LIN {X 0,Y 474.618,Z 150.861,A -85,B 0,C 180,E1 -7365.42,E2 -7365.42} C_VEL
LIN {X 0,Y 474.69,Z 150.851,A -85,B 0,C 180,E1 -7368.037,E2 -7368.037} C_VEL
LIN {X 0,Y 474.695,Z 150.851,A -85,B 0,C 180,E1 -7371.486,E2 -7371.486} C_VEL
LIN {X 0,Y 474.744,Z 150.845,A -85,B 0,C 180,E1 -7374.052,E2 -7374.052} C_VEL
LIN {X 0,Y 474.866,Z 150.829,A -85,B 0,C 180,E1 -7377.455,E2 -7377.455} C_VEL
LIN {X 0,Y 474.862,Z 150.83,A -85,B 0,C 180,E1 -7380,E2 -7380} C_VEL
LIN {X 0,Y 474.862,Z 150.835,A -85,B 0,C 180,E1 -7382.544,E2 -7382.544} C_VEL
LIN {X 0,Y 474.742,Z 150.847,A -85,B 0,C 180,E1 -7385.948,E2 -7385.948} C_VEL
LIN {X 0,Y 474.685,Z 150.857,A -85,B 0,C 180,E1 -7388.514,E2 -7388.514} C_VEL
LIN {X 0,Y 474.677,Z 150.856,A -85,B 0,C 180,E1 -7391.963,E2 -7391.963} C_VEL
LIN {X 0,Y 474.683,Z 150.854,A -85,B 0,C 180,E1 -7395.456,E2 -7395.456} C_VEL
LIN {X 0,Y 474.646,Z 150.859,A -85,B 0,C 180,E1 -7399.011,E2 -7399.011} C_VEL
LIN {X 0,Y 474.574,Z 150.87,A -85,B 0,C 180,E1 -7401.729,E2 -7401.729} C_VEL
LIN {X 0,Y 474.611,Z 150.865,A -85,B 0,C 180,E1 -7404.495,E2 -7404.495} C_VEL
LIN {X 0,Y 474.583,Z 150.867,A -85,B 0,C 180,E1 -7407.327,E2 -7407.327} C_VEL
LIN {X 0,Y 474.596,Z 150.87,A -85,B 0,C 180,E1 -7410.23,E2 -7410.23} C_VEL
LIN {X 0,Y 474.648,Z 151.03,A -85,B 0,C 180,E1 -7411.586,E2 -7411.586} C_VEL
LIN {X 0,Y 475.967,Z 158.401,A -85,B 0,C 180,E1 -7413.115,E2 -7413.115} C_VEL
LIN {X 0,Y 475.697,Z 171.558,A -85,B 0,C 180,E1 -7415.654,E2 -7415.654} C_VEL
LIN {X 0,Y 475.449,Z 180.026,A -85,B 0,C 180,E1 -7417.232,E2 -7417.232} C_VEL
LIN {X 0,Y 476.208,Z 184.236,A -85,B 0,C 180,E1 -7417.368,E2 -7417.368} C_VEL
LIN {X 0,Y 478.194,Z 196.098,A -85,B 0,C 180,E1 -7417.633,E2 -7417.633} C_VEL
LIN {X 0,Y 477.381,Z 287.664,A -85,B 0,C 180,E1 -7419.069,E2 -7419.069} C_VEL
LIN {X 0,Y 477.141,Z 300.656,A -85,B 0,C 180,E1 -7419.44,E2 -7419.44} C_VEL
LIN {X 0,Y 476.759,Z 313.013,A -85,B 0,C 180,E1 -7419.958,E2 -7419.958} C_VEL
LIN {X 0,Y 476.372,Z 324.473,A -85,B 0,C 180,E1 -7420.606,E2 -7420.606} C_VEL
LIN {X 0,Y 475.88,Z 335.964,A -85,B 0,C 180,E1 -7421.447,E2 -7421.447} C_VEL
LIN {X 0,Y 475.436,Z 345.842,A -85,B 0,C 180,E1 -7422.347,E2 -7422.347} C_VEL
LIN {X 0,Y 475.017,Z 354.974,A -85,B 0,C 180,E1 -7423.363,E2 -7423.363} C_VEL
LIN {X 0,Y 474.602,Z 363.651,A -85,B 0,C 180,E1 -7424.545,E2 -7424.545} C_VEL
LIN {X 0,Y 474.265,Z 371.371,A -85,B 0,C 180,E1 -7425.857,E2 -7425.857} C_VEL
LIN {X 0,Y 474.065,Z 376.86,A -85,B 0,C 180,E1 -7427.006,E2 -7427.006} C_VEL
LIN {X 0,Y 473.921,Z 381.283,A -85,B 0,C 180,E1 -7428.141,E2 -7428.141} C_VEL
LIN {X 0,Y 473.859,Z 384.78,A -85,B 0,C 180,E1 -7429.265,E2 -7429.265} C_VEL
LIN {X 0,Y 473.679,Z 387.66,A -85,B 0,C 180,E1 -7430.49,E2 -7430.49} C_VEL
LIN {X 0,Y 473.595,Z 389.84,A -85,B 0,C 180,E1 -7431.859,E2 -7431.859} C_VEL
LIN {X 0,Y 473.572,Z 390.497,A -85,B 0,C 180,E1 -7432.508,E2 -7432.508} C_VEL
LIN {X 0,Y 472.915,Z 391.073,A -85,B 0,C 180,E1 -7433.216,E2 -7433.216} C_VEL
LIN {X 0,Y 470.061,Z 391.361,A -85,B 0,C 180,E1 -7434.371,E2 -7434.371} C_VEL
LIN {X 0,Y 467.642,Z 390.943,A -85,B 0,C 180,E1 -7435.301,E2 -7435.301} C_VEL
LIN {X 0,Y 466.601,Z 390.22,A -85,B 0,C 180,E1 -7436.015,E2 -7436.015} C_VEL
LIN {X 0,Y 466.515,Z 389.897,A -85,B 0,C 180,E1 -7436.255,E2 -7436.255} C_VEL
LIN {X 0,Y 466.607,Z 387.998,A -85,B 0,C 180,E1 -7437.507,E2 -7437.507} C_VEL
LIN {X 0,Y 466.734,Z 384.141,A -85,B 0,C 180,E1 -7439.125,E2 -7439.125} C_VEL
LIN {X 0,Y 466.909,Z 379.431,A -85,B 0,C 180,E1 -7440.543,E2 -7440.543} C_VEL
LIN {X 0,Y 467.152,Z 373.328,A -85,B 0,C 180,E1 -7441.958,E2 -7441.958} C_VEL
LIN {X 0,Y 467.413,Z 366.653,A -85,B 0,C 180,E1 -7443.189,E2 -7443.189} C_VEL
LIN {X 0,Y 467.847,Z 357.754,A -85,B 0,C 180,E1 -7444.505,E2 -7444.505} C_VEL
LIN {X 0,Y 468.279,Z 348.414,A -85,B 0,C 180,E1 -7445.625,E2 -7445.625} C_VEL
LIN {X 0,Y 468.758,Z 338.491,A -85,B 0,C 180,E1 -7446.591,E2 -7446.591} C_VEL
LIN {X 0,Y 469.247,Z 327.717,A -85,B 0,C 180,E1 -7447.433,E2 -7447.433} C_VEL
LIN {X 0,Y 469.72,Z 315.436,A -85,B 0,C 180,E1 -7448.185,E2 -7448.185} C_VEL
LIN {X 0,Y 470.111,Z 303.17,A -85,B 0,C 180,E1 -7448.746,E2 -7448.746} C_VEL
LIN {X 0,Y 470.403,Z 289.73,A -85,B 0,C 180,E1 -7449.161,E2 -7449.161} C_VEL
LIN {X 0,Y 470.644,Z 267.567,A -85,B 0,C 180,E1 -7449.543,E2 -7449.543} C_VEL
LIN {X 0,Y 471.141,Z 195.55,A -85,B 0,C 180,E1 -7450.672,E2 -7450.672} C_VEL
LIN {X 0,Y 468.481,Z 180.547,A -85,B 0,C 180,E1 -7451.028,E2 -7451.028} C_VEL
LIN {X 0,Y 468.525,Z 177.121,A -85,B 0,C 180,E1 -7451.64,E2 -7451.64} C_VEL
LIN {X 0,Y 469.221,Z 161.481,A -85,B 0,C 180,E1 -7454.806,E2 -7454.806} C_VEL
LIN {X 0,Y 468.327,Z 155.391,A -85,B 0,C 180,E1 -7456.108,E2 -7456.108} C_VEL
LIN {X 0,Y 467.639,Z 151.805,A -85,B 0,C 180,E1 -7456.945,E2 -7456.945} C_VEL
LIN {X 0,Y 467.624,Z 151.736,A -85,B 0,C 180,E1 -7459.611,E2 -7459.611} C_VEL
LIN {X 0,Y 467.749,Z 151.716,A -85,B 0,C 180,E1 -7462.591,E2 -7462.591} C_VEL
LIN {X 0,Y 467.721,Z 151.719,A -85,B 0,C 180,E1 -7464.828,E2 -7464.828} C_VEL
LIN {X 0,Y 467.856,Z 151.705,A -85,B 0,C 180,E1 -7467.418,E2 -7467.418} C_VEL
LIN {X 0,Y 467.879,Z 151.704,A -85,B 0,C 180,E1 -7470.001,E2 -7470.001} C_VEL
LIN {X 0,Y 467.856,Z 151.702,A -85,B 0,C 180,E1 -7472.584,E2 -7472.584} C_VEL
LIN {X 0,Y 467.732,Z 151.721,A -85,B 0,C 180,E1 -7476.038,E2 -7476.038} C_VEL
LIN {X 0,Y 467.669,Z 151.726,A -85,B 0,C 180,E1 -7478.644,E2 -7478.644} C_VEL
LIN {X 0,Y 467.655,Z 151.728,A -85,B 0,C 180,E1 -7482.146,E2 -7482.146} C_VEL
LIN {X 0,Y 467.638,Z 151.734,A -85,B 0,C 180,E1 -7485.696,E2 -7485.696} C_VEL
LIN {X 0,Y 467.621,Z 151.74,A -85,B 0,C 180,E1 -7489.308,E2 -7489.308} C_VEL
LIN {X 0,Y 467.533,Z 151.743,A -85,B 0,C 180,E1 -7492.075,E2 -7492.075} C_VEL
LIN {X 0,Y 467.584,Z 151.74,A -85,B 0,C 180,E1 -7494.889,E2 -7494.889} C_VEL
LIN {X 0,Y 467.618,Z 151.733,A -85,B 0,C 180,E1 -7497.77,E2 -7497.77} C_VEL
LIN {X 0,Y 467.566,Z 151.746,A -85,B 0,C 180,E1 -7501.045,E2 -7501.045} C_VEL
LIN {X 0,Y 467.576,Z 151.738,A -85,B 0,C 180,E1 -7504.241,E2 -7504.241} C_VEL
LIN {X 0,Y 467.547,Z 151.746,A -85,B 0,C 180,E1 -7507.187,E2 -7507.187} C_VEL
LIN {X 0,Y 467.573,Z 151.739,A -85,B 0,C 180,E1 -7510.265,E2 -7510.265} C_VEL
LIN {X 0,Y 467.586,Z 151.741,A -85,B 0,C 180,E1 -7512.567,E2 -7512.567} C_VEL
LIN {X 0,Y 467.565,Z 151.743,A -85,B 0,C 180,E1 -7515.053,E2 -7515.053} C_VEL
LIN {X 0,Y 467.572,Z 151.745,A -85,B 0,C 180,E1 -7518.597,E2 -7518.597} C_VEL
LIN {X 0,Y 467.561,Z 151.74,A -85,B 0,C 180,E1 -7521.956,E2 -7521.956} C_VEL
LIN {X 0,Y 467.561,Z 151.74,A -85,B 0,C 180,E1 -7525.168,E2 -7525.168} C_VEL
LIN {X 0,Y 467.582,Z 151.742,A -85,B 0,C 180,E1 -7528.26,E2 -7528.26} C_VEL
LIN {X 0,Y 467.554,Z 151.74,A -85,B 0,C 180,E1 -7531.249,E2 -7531.249} C_VEL
LIN {X 0,Y 467.582,Z 151.742,A -85,B 0,C 180,E1 -7534.159,E2 -7534.159} C_VEL
LIN {X 0,Y 467.575,Z 151.738,A -85,B 0,C 180,E1 -7536.996,E2 -7536.996} C_VEL
LIN {X 0,Y 467.621,Z 151.734,A -85,B 0,C 180,E1 -7539.778,E2 -7539.778} C_VEL
LIN {X 0,Y 467.593,Z 151.739,A -85,B 0,C 180,E1 -7542.507,E2 -7542.507} C_VEL
LIN {X 0,Y 467.599,Z 151.734,A -85,B 0,C 180,E1 -7545.197,E2 -7545.197} C_VEL
LIN {X 0,Y 467.656,Z 151.733,A -85,B 0,C 180,E1 -7547.855,E2 -7547.855} C_VEL
LIN {X 0,Y 467.657,Z 151.728,A -85,B 0,C 180,E1 -7551.357,E2 -7551.357} C_VEL
LIN {X 0,Y 467.702,Z 151.729,A -85,B 0,C 180,E1 -7553.962,E2 -7553.962} C_VEL
LIN {X 0,Y 467.813,Z 151.71,A -85,B 0,C 180,E1 -7557.417,E2 -7557.417} C_VEL
LIN {X 0,Y 467.848,Z 151.708,A -85,B 0,C 180,E1 -7560,E2 -7560} C_VEL
LIN {X 0,Y 467.822,Z 151.707,A -85,B 0,C 180,E1 -7562.583,E2 -7562.583} C_VEL
LIN {X 0,Y 467.694,Z 151.726,A -85,B 0,C 180,E1 -7566.038,E2 -7566.038} C_VEL
LIN {X 0,Y 467.636,Z 151.73,A -85,B 0,C 180,E1 -7568.644,E2 -7568.644} C_VEL
LIN {X 0,Y 467.656,Z 151.728,A -85,B 0,C 180,E1 -7572.146,E2 -7572.146} C_VEL
LIN {X 0,Y 467.638,Z 151.734,A -85,B 0,C 180,E1 -7575.695,E2 -7575.695} C_VEL
LIN {X 0,Y 467.617,Z 151.74,A -85,B 0,C 180,E1 -7579.308,E2 -7579.308} C_VEL
LIN {X 0,Y 467.53,Z 151.743,A -85,B 0,C 180,E1 -7582.074,E2 -7582.074} C_VEL
LIN {X 0,Y 467.551,Z 151.744,A -85,B 0,C 180,E1 -7584.891,E2 -7584.891} C_VEL
LIN {X 0,Y 467.538,Z 151.743,A -85,B 0,C 180,E1 -7587.775,E2 -7587.775} C_VEL
LIN {X 0,Y 467.528,Z 151.75,A -85,B 0,C 180,E1 -7591.036,E2 -7591.036} C_VEL
LIN {X 0,Y 467.566,Z 151.739,A -85,B 0,C 180,E1 -7594.238,E2 -7594.238} C_VEL
LIN {X 0,Y 467.517,Z 151.75,A -85,B 0,C 180,E1 -7597.181,E2 -7597.181} C_VEL
LIN {X 0,Y 467.519,Z 151.745,A -85,B 0,C 180,E1 -7600.271,E2 -7600.271} C_VEL
LIN {X 0,Y 467.518,Z 151.749,A -85,B 0,C 180,E1 -7602.569,E2 -7602.569} C_VEL
LIN {X 0,Y 467.564,Z 151.743,A -85,B 0,C 180,E1 -7605.052,E2 -7605.052} C_VEL
LIN {X 0,Y 467.552,Z 151.748,A -85,B 0,C 180,E1 -7608.727,E2 -7608.727} C_VEL
LIN {X 0,Y 467.533,Z 151.743,A -85,B 0,C 180,E1 -7611.952,E2 -7611.952} C_VEL
LIN {X 0,Y 467.511,Z 151.747,A -85,B 0,C 180,E1 -7615.162,E2 -7615.162} C_VEL
LIN {X 0,Y 467.544,Z 151.746,A -85,B 0,C 180,E1 -7618.256,E2 -7618.256} C_VEL
LIN {X 0,Y 467.527,Z 151.747,A -85,B 0,C 180,E1 -7621.247,E2 -7621.247} C_VEL
LIN {X 0,Y 467.571,Z 151.743,A -85,B 0,C 180,E1 -7624.693,E2 -7624.693} C_VEL
LIN {X 0,Y 467.652,Z 152.044,A -85,B 0,C 180,E1 -7625.063,E2 -7625.063} C_VEL
LIN {X 0,Y 469.67,Z 163.271,A -85,B 0,C 180,E1 -7627.336,E2 -7627.336} C_VEL
LIN {X 0,Y 469.027,Z 176.652,A -85,B 0,C 180,E1 -7629.84,E2 -7629.84} C_VEL
LIN {X 0,Y 468.4,Z 193.099,A -85,B 0,C 180,E1 -7632.874,E2 -7632.874} C_VEL
LIN {X 0,Y 468.424,Z 194.305,A -85,B 0,C 180,E1 -7633.012,E2 -7633.012} C_VEL
LIN {X 0,Y 471.201,Z 212.37,A -85,B 0,C 180,E1 -7633.414,E2 -7633.414} C_VEL
LIN {X 0,Y 470.448,Z 302.366,A -85,B 0,C 180,E1 -7634.844,E2 -7634.844} C_VEL
LIN {X 0,Y 470.115,Z 316.1,A -85,B 0,C 180,E1 -7635.249,E2 -7635.249} C_VEL
LIN {X 0,Y 469.595,Z 328.968,A -85,B 0,C 180,E1 -7635.813,E2 -7635.813} C_VEL
LIN {X 0,Y 469.143,Z 341.516,A -85,B 0,C 180,E1 -7636.573,E2 -7636.573} C_VEL
LIN {X 0,Y 468.697,Z 351.766,A -85,B 0,C 180,E1 -7637.361,E2 -7637.361} C_VEL
LIN {X 0,Y 468.243,Z 361.774,A -85,B 0,C 180,E1 -7638.309,E2 -7638.309} C_VEL
LIN {X 0,Y 467.76,Z 371.066,A -85,B 0,C 180,E1 -7639.393,E2 -7639.393} C_VEL
LIN {X 0,Y 467.349,Z 380.084,A -85,B 0,C 180,E1 -7640.696,E2 -7640.696} C_VEL
LIN {X 0,Y 467.045,Z 387.346,A -85,B 0,C 180,E1 -7641.998,E2 -7641.998} C_VEL
LIN {X 0,Y 466.851,Z 392.246,A -85,B 0,C 180,E1 -7643.082,E2 -7643.082} C_VEL
LIN {X 0,Y 466.789,Z 397.007,A -85,B 0,C 180,E1 -7644.383,E2 -7644.383} C_VEL
LIN {X 0,Y 466.647,Z 400.642,A -85,B 0,C 180,E1 -7645.681,E2 -7645.681} C_VEL
LIN {X 0,Y 466.661,Z 402.52,A -85,B 0,C 180,E1 -7646.546,E2 -7646.546} C_VEL
LIN {X 0,Y 466.645,Z 403.929,A -85,B 0,C 180,E1 -7647.41,E2 -7647.41} C_VEL
LIN {X 0,Y 466.59,Z 405.543,A -85,B 0,C 180,E1 -7649.136,E2 -7649.136} C_VEL
LIN {X 0,Y 466.599,Z 405.763,A -85,B 0,C 180,E1 -7649.999,E2 -7649.999} C_VEL
LIN {X 0,Y 466.59,Z 405.549,A -85,B 0,C 180,E1 -7650.862,E2 -7650.862} C_VEL
LIN {X 0,Y 466.644,Z 403.941,A -85,B 0,C 180,E1 -7652.589,E2 -7652.589} C_VEL
LIN {X 0,Y 466.66,Z 402.54,A -85,B 0,C 180,E1 -7653.453,E2 -7653.453} C_VEL
LIN {X 0,Y 466.691,Z 399.593,A -85,B 0,C 180,E1 -7654.75,E2 -7654.75} C_VEL
LIN {X 0,Y 466.778,Z 395.605,A -85,B 0,C 180,E1 -7656.049,E2 -7656.049} C_VEL
LIN {X 0,Y 466.976,Z 389.468,A -85,B 0,C 180,E1 -7657.566,E2 -7657.566} C_VEL
LIN {X 0,Y 467.25,Z 382.762,A -85,B 0,C 180,E1 -7658.868,E2 -7658.868} C_VEL
LIN {X 0,Y 467.596,Z 374.442,A -85,B 0,C 180,E1 -7660.171,E2 -7660.171} C_VEL
LIN {X 0,Y 468.048,Z 365.905,A -85,B 0,C 180,E1 -7661.255,E2 -7661.255} C_VEL
LIN {X 0,Y 468.546,Z 355.648,A -85,B 0,C 180,E1 -7662.314,E2 -7662.314} C_VEL
LIN {X 0,Y 468.965,Z 345.212,A -85,B 0,C 180,E1 -7663.188,E2 -7663.188} C_VEL
LIN {X 0,Y 469.469,Z 333.466,A -85,B 0,C 180,E1 -7663.968,E2 -7663.968} C_VEL
LIN {X 0,Y 470.027,Z 320.332,A -85,B 0,C 180,E1 -7664.614,E2 -7664.614} C_VEL
LIN {X 0,Y 470.38,Z 307.097,A -85,B 0,C 180,E1 -7665.073,E2 -7665.073} C_VEL
LIN {X 0,Y 470.645,Z 294.151,A -85,B 0,C 180,E1 -7665.341,E2 -7665.341} C_VEL
LIN {X 0,Y 471.224,Z 210.985,A -85,B 0,C 180,E1 -7666.652,E2 -7666.652} C_VEL
LIN {X 0,Y 468.452,Z 193.768,A -85,B 0,C 180,E1 -7667.059,E2 -7667.059} C_VEL
LIN {X 0,Y 468.76,Z 184.094,A -85,B 0,C 180,E1 -7668.766,E2 -7668.766} C_VEL
LIN {X 0,Y 469.551,Z 165.471,A -85,B 0,C 180,E1 -7672.204,E2 -7672.204} C_VEL
LIN {X 0,Y 469.274,Z 160.557,A -85,B 0,C 180,E1 -7673.148,E2 -7673.148} C_VEL
LIN {X 0,Y 467.617,Z 151.879,A -85,B 0,C 180,E1 -7674.937,E2 -7674.937} C_VEL
LIN {X 0,Y 467.535,Z 151.748,A -85,B 0,C 180,E1 -7677.773,E2 -7677.773} C_VEL
LIN {X 0,Y 467.525,Z 151.748,A -85,B 0,C 180,E1 -7681.035,E2 -7681.035} C_VEL
LIN {X 0,Y 467.561,Z 151.746,A -85,B 0,C 180,E1 -7683.789,E2 -7683.789} C_VEL
LIN {X 0,Y 467.496,Z 151.751,A -85,B 0,C 180,E1 -7686.963,E2 -7686.963} C_VEL
LIN {X 0,Y 467.553,Z 151.743,A -85,B 0,C 180,E1 -7689.95,E2 -7689.95} C_VEL
LIN {X 0,Y 467.509,Z 151.747,A -85,B 0,C 180,E1 -7692.567,E2 -7692.567} C_VEL
LIN {X 0,Y 467.554,Z 151.745,A -85,B 0,C 180,E1 -7695.051,E2 -7695.051} C_VEL
LIN {X 0,Y 467.551,Z 151.744,A -85,B 0,C 180,E1 -7698.725,E2 -7698.725} C_VEL
LIN {X 0,Y 467.537,Z 151.741,A -85,B 0,C 180,E1 -7701.952,E2 -7701.952} C_VEL
LIN {X 0,Y 467.545,Z 151.745,A -85,B 0,C 180,E1 -7705.165,E2 -7705.165} C_VEL
LIN {X 0,Y 467.537,Z 151.742,A -85,B 0,C 180,E1 -7708.256,E2 -7708.256} C_VEL
LIN {X 0,Y 467.529,Z 151.748,A -85,B 0,C 180,E1 -7711.247,E2 -7711.247} C_VEL
LIN {X 0,Y 467.564,Z 151.74,A -85,B 0,C 180,E1 -7714.4,E2 -7714.4} C_VEL
LIN {X 0,Y 467.56,Z 151.742,A -85,B 0,C 180,E1 -7716.995,E2 -7716.995} C_VEL
LIN {X 0,Y 467.607,Z 151.732,A -85,B 0,C 180,E1 -7719.776,E2 -7719.776} C_VEL
LIN {X 0,Y 467.58,Z 151.739,A -85,B 0,C 180,E1 -7722.505,E2 -7722.505} C_VEL
LIN {X 0,Y 467.58,Z 151.739,A -85,B 0,C 180,E1 -7725.195,E2 -7725.195} C_VEL
LIN {X 0,Y 467.642,Z 151.729,A -85,B 0,C 180,E1 -7727.854,E2 -7727.854} C_VEL
LIN {X 0,Y 467.653,Z 151.729,A -85,B 0,C 180,E1 -7731.356,E2 -7731.356} C_VEL
LIN {X 0,Y 467.709,Z 151.721,A -85,B 0,C 180,E1 -7733.962,E2 -7733.962} C_VEL
LIN {X 0,Y 467.807,Z 151.709,A -85,B 0,C 180,E1 -7737.416,E2 -7737.416} C_VEL
LIN {X 0,Y 467.832,Z 151.706,A -85,B 0,C 180,E1 -7740,E2 -7740} C_VEL
LIN {X 0,Y 467.803,Z 151.714,A -85,B 0,C 180,E1 -7742.583,E2 -7742.583} C_VEL
LIN {X 0,Y 467.707,Z 151.725,A -85,B 0,C 180,E1 -7746.037,E2 -7746.037} C_VEL
LIN {X 0,Y 467.644,Z 151.733,A -85,B 0,C 180,E1 -7748.643,E2 -7748.643} C_VEL
LIN {X 0,Y 467.633,Z 151.737,A -85,B 0,C 180,E1 -7752.353,E2 -7752.353} C_VEL
LIN {X 0,Y 467.634,Z 151.734,A -85,B 0,C 180,E1 -7755.885,E2 -7755.885} C_VEL
LIN {X 0,Y 467.605,Z 151.735,A -85,B 0,C 180,E1 -7759.308,E2 -7759.308} C_VEL
LIN {X 0,Y 467.52,Z 151.752,A -85,B 0,C 180,E1 -7762.074,E2 -7762.074} C_VEL
LIN {X 0,Y 467.541,Z 151.742,A -85,B 0,C 180,E1 -7764.89,E2 -7764.89} C_VEL
LIN {X 0,Y 467.53,Z 151.75,A -85,B 0,C 180,E1 -7767.774,E2 -7767.774} C_VEL
LIN {X 0,Y 467.592,Z 151.77,A -85,B 0,C 180,E1 -7771.304,E2 -7771.304} C_VEL
LIN {X 0,Y 467.91,Z 153.38,A -85,B 0,C 180,E1 -7771.715,E2 -7771.715} C_VEL
LIN {X 0,Y 469.117,Z 160.695,A -85,B 0,C 180,E1 -7773.227,E2 -7773.227} C_VEL
LIN {X 0,Y 468.577,Z 176.798,A -85,B 0,C 180,E1 -7776.358,E2 -7776.358} C_VEL
LIN {X 0,Y 468.497,Z 180.374,A -85,B 0,C 180,E1 -7776.99,E2 -7776.99} C_VEL
LIN {X 0,Y 471.401,Z 196.938,A -85,B 0,C 180,E1 -7777.396,E2 -7777.396} C_VEL
LIN {X 0,Y 470.529,Z 288.212,A -85,B 0,C 180,E1 -7778.853,E2 -7778.853} C_VEL
LIN {X 0,Y 470.261,Z 301.569,A -85,B 0,C 180,E1 -7779.247,E2 -7779.247} C_VEL
LIN {X 0,Y 469.863,Z 313.653,A -85,B 0,C 180,E1 -7779.769,E2 -7779.769} C_VEL
LIN {X 0,Y 469.465,Z 325.059,A -85,B 0,C 180,E1 -7780.434,E2 -7780.434} C_VEL
LIN {X 0,Y 468.946,Z 336.085,A -85,B 0,C 180,E1 -7781.255,E2 -7781.255} C_VEL
LIN {X 0,Y 468.438,Z 347.001,A -85,B 0,C 180,E1 -7782.274,E2 -7782.274} C_VEL
LIN {X 0,Y 467.954,Z 356.383,A -85,B 0,C 180,E1 -7783.361,E2 -7783.361} C_VEL
LIN {X 0,Y 467.575,Z 364.05,A -85,B 0,C 180,E1 -7784.444,E2 -7784.444} C_VEL
LIN {X 0,Y 467.251,Z 370.927,A -85,B 0,C 180,E1 -7785.622,E2 -7785.622} C_VEL
LIN {X 0,Y 466.978,Z 377.764,A -85,B 0,C 180,E1 -7787.086,E2 -7787.086} C_VEL
LIN {X 0,Y 466.812,Z 382.933,A -85,B 0,C 180,E1 -7788.516,E2 -7788.516} C_VEL
LIN {X 0,Y 466.732,Z 386.048,A -85,B 0,C 180,E1 -7789.649,E2 -7789.649} C_VEL
LIN {X 0,Y 466.551,Z 388.371,A -85,B 0,C 180,E1 -7790.754,E2 -7790.754} C_VEL
LIN {X 0,Y 466.501,Z 389.994,A -85,B 0,C 180,E1 -7791.855,E2 -7791.855} C_VEL
LIN {X 0,Y 466.464,Z 390.951,A -85,B 0,C 180,E1 -7792.989,E2 -7792.989} C_VEL
LIN {X 0,Y 466.473,Z 391.191,A -85,B 0,C 180,E1 -7794.446,E2 -7794.446} C_VEL
LIN {X 0,Y 466.518,Z 390.082,A -85,B 0,C 180,E1 -7796.126,E2 -7796.126} C_VEL
LIN {X 0,Y 466.515,Z 389.897,A -85,B 0,C 180,E1 -7796.255,E2 -7796.255} C_VEL
LIN {X 0,Y 465.857,Z 388.944,A -85,B 0,C 180,E1 -7796.965,E2 -7796.965} C_VEL
LIN {X 0,Y 463.07,Z 386.859,A -85,B 0,C 180,E1 -7798.112,E2 -7798.112} C_VEL
LIN {X 0,Y 460.751,Z 384.699,A -85,B 0,C 180,E1 -7799.022,E2 -7799.022} C_VEL
LIN {X 0,Y 459.803,Z 382.722,A -85,B 0,C 180,E1 -7799.711,E2 -7799.711} C_VEL
LIN {X 0,Y 459.75,Z 381.978,A -85,B 0,C 180,E1 -7799.94,E2 -7799.94} C_VEL
LIN {X 0,Y 459.973,Z 376.142,A -85,B 0,C 180,E1 -7801.481,E2 -7801.481} C_VEL
LIN {X 0,Y 460.246,Z 370.049,A -85,B 0,C 180,E1 -7802.737,E2 -7802.737} C_VEL
LIN {X 0,Y 460.611,Z 362.499,A -85,B 0,C 180,E1 -7803.996,E2 -7803.996} C_VEL
LIN {X 0,Y 461.063,Z 353.471,A -85,B 0,C 180,E1 -7805.218,E2 -7805.218} C_VEL
LIN {X 0,Y 461.576,Z 343.75,A -85,B 0,C 180,E1 -7806.289,E2 -7806.289} C_VEL
LIN {X 0,Y 462.054,Z 333.759,A -85,B 0,C 180,E1 -7807.18,E2 -7807.18} C_VEL
LIN {X 0,Y 462.601,Z 321.462,A -85,B 0,C 180,E1 -7808.046,E2 -7808.046} C_VEL
LIN {X 0,Y 463.049,Z 309.37,A -85,B 0,C 180,E1 -7808.697,E2 -7808.697} C_VEL
LIN {X 0,Y 463.416,Z 296.417,A -85,B 0,C 180,E1 -7809.195,E2 -7809.195} C_VEL
LIN {X 0,Y 463.685,Z 282.639,A -85,B 0,C 180,E1 -7809.527,E2 -7809.527} C_VEL
LIN {X 0,Y 464.294,Z 196.146,A -85,B 0,C 180,E1 -7810.906,E2 -7810.906} C_VEL
LIN {X 0,Y 461.519,Z 180.623,A -85,B 0,C 180,E1 -7811.284,E2 -7811.284} C_VEL
LIN {X 0,Y 461.634,Z 176.516,A -85,B 0,C 180,E1 -7812.045,E2 -7812.045} C_VEL
LIN {X 0,Y 462.238,Z 162.044,A -85,B 0,C 180,E1 -7815.022,E2 -7815.022} C_VEL
LIN {X 0,Y 460.603,Z 152.734,A -85,B 0,C 180,E1 -7817.107,E2 -7817.107} C_VEL
LIN {X 0,Y 460.61,Z 152.61,A -85,B 0,C 180,E1 -7820.339,E2 -7820.339} C_VEL
LIN {X 0,Y 460.669,Z 152.598,A -85,B 0,C 180,E1 -7822.991,E2 -7822.991} C_VEL
LIN {X 0,Y 460.694,Z 152.595,A -85,B 0,C 180,E1 -7824.749,E2 -7824.749} C_VEL
LIN {X 0,Y 460.797,Z 152.584,A -85,B 0,C 180,E1 -7827.378,E2 -7827.378} C_VEL
LIN {X 0,Y 460.849,Z 152.58,A -85,B 0,C 180,E1 -7830.001,E2 -7830.001} C_VEL
LIN {X 0,Y 460.797,Z 152.582,A -85,B 0,C 180,E1 -7832.623,E2 -7832.623} C_VEL
LIN {X 0,Y 460.697,Z 152.596,A -85,B 0,C 180,E1 -7836.131,E2 -7836.131} C_VEL
LIN {X 0,Y 460.619,Z 152.604,A -85,B 0,C 180,E1 -7838.777,E2 -7838.777} C_VEL
LIN {X 0,Y 460.612,Z 152.605,A -85,B 0,C 180,E1 -7842.446,E2 -7842.446} C_VEL
LIN {X 0,Y 460.599,Z 152.608,A -85,B 0,C 180,E1 -7845.998,E2 -7845.998} C_VEL
LIN {X 0,Y 460.567,Z 152.614,A -85,B 0,C 180,E1 -7849.616,E2 -7849.616} C_VEL
LIN {X 0,Y 460.509,Z 152.618,A -85,B 0,C 180,E1 -7852.429,E2 -7852.429} C_VEL
LIN {X 0,Y 460.552,Z 152.613,A -85,B 0,C 180,E1 -7855.799,E2 -7855.799} C_VEL
LIN {X 0,Y 460.55,Z 152.612,A -85,B 0,C 180,E1 -7858.234,E2 -7858.234} C_VEL
LIN {X 0,Y 460.519,Z 152.621,A -85,B 0,C 180,E1 -7861.283,E2 -7861.283} C_VEL
LIN {X 0,Y 460.522,Z 152.618,A -85,B 0,C 180,E1 -7864.504,E2 -7864.504} C_VEL
LIN {X 0,Y 460.5,Z 152.619,A -85,B 0,C 180,E1 -7867.624,E2 -7867.624} C_VEL
LIN {X 0,Y 460.537,Z 152.615,A -85,B 0,C 180,E1 -7870.269,E2 -7870.269} C_VEL
LIN {X 0,Y 460.498,Z 152.62,A -85,B 0,C 180,E1 -7873.376,E2 -7873.376} C_VEL
LIN {X 0,Y 460.508,Z 152.624,A -85,B 0,C 180,E1 -7876.626,E2 -7876.626} C_VEL
LIN {X 0,Y 460.534,Z 152.614,A -85,B 0,C 180,E1 -7879.732,E2 -7879.732} C_VEL
LIN {X 0,Y 460.496,Z 152.626,A -85,B 0,C 180,E1 -7882.525,E2 -7882.525} C_VEL
LIN {X 0,Y 460.544,Z 152.613,A -85,B 0,C 180,E1 -7885.624,E2 -7885.624} C_VEL
LIN {X 0,Y 460.537,Z 152.618,A -85,B 0,C 180,E1 -7888.745,E2 -7888.745} C_VEL
LIN {X 0,Y 460.55,Z 152.619,A -85,B 0,C 180,E1 -7892.262,E2 -7892.262} C_VEL
LIN {X 0,Y 460.534,Z 152.618,A -85,B 0,C 180,E1 -7894.704,E2 -7894.704} C_VEL
LIN {X 0,Y 460.509,Z 152.618,A -85,B 0,C 180,E1 -7897.572,E2 -7897.572} C_VEL
LIN {X 0,Y 460.567,Z 152.616,A -85,B 0,C 180,E1 -7900.385,E2 -7900.385} C_VEL
LIN {X 0,Y 460.605,Z 152.613,A -85,B 0,C 180,E1 -7904.059,E2 -7904.059} C_VEL
LIN {X 0,Y 460.609,Z 152.608,A -85,B 0,C 180,E1 -7907.666,E2 -7907.666} C_VEL
LIN {X 0,Y 460.609,Z 152.605,A -85,B 0,C 180,E1 -7911.224,E2 -7911.224} C_VEL
LIN {X 0,Y 460.668,Z 152.605,A -85,B 0,C 180,E1 -7913.87,E2 -7913.87} C_VEL
LIN {X 0,Y 460.757,Z 152.589,A -85,B 0,C 180,E1 -7917.378,E2 -7917.378} C_VEL
LIN {X 0,Y 460.818,Z 152.584,A -85,B 0,C 180,E1 -7920,E2 -7920} C_VEL
LIN {X 0,Y 460.767,Z 152.585,A -85,B 0,C 180,E1 -7922.623,E2 -7922.623} C_VEL
LIN {X 0,Y 460.66,Z 152.601,A -85,B 0,C 180,E1 -7926.131,E2 -7926.131} C_VEL
LIN {X 0,Y 460.591,Z 152.608,A -85,B 0,C 180,E1 -7928.777,E2 -7928.777} C_VEL
LIN {X 0,Y 460.61,Z 152.605,A -85,B 0,C 180,E1 -7932.335,E2 -7932.335} C_VEL
LIN {X 0,Y 460.58,Z 152.61,A -85,B 0,C 180,E1 -7935.988,E2 -7935.988} C_VEL
LIN {X 0,Y 460.562,Z 152.615,A -85,B 0,C 180,E1 -7939.616,E2 -7939.616} C_VEL
LIN {X 0,Y 460.507,Z 152.618,A -85,B 0,C 180,E1 -7942.429,E2 -7942.429} C_VEL
LIN {X 0,Y 460.511,Z 152.625,A -85,B 0,C 180,E1 -7945.298,E2 -7945.298} C_VEL
LIN {X 0,Y 460.496,Z 152.619,A -85,B 0,C 180,E1 -7948.237,E2 -7948.237} C_VEL
LIN {X 0,Y 460.497,Z 152.625,A -85,B 0,C 180,E1 -7951.278,E2 -7951.278} C_VEL
LIN {X 0,Y 460.513,Z 152.619,A -85,B 0,C 180,E1 -7954.502,E2 -7954.502} C_VEL
LIN {X 0,Y 460.484,Z 152.622,A -85,B 0,C 180,E1 -7957.625,E2 -7957.625} C_VEL
LIN {X 0,Y 460.501,Z 152.625,A -85,B 0,C 180,E1 -7961.015,E2 -7961.015} C_VEL
LIN {X 0,Y 460.512,Z 152.622,A -85,B 0,C 180,E1 -7964.59,E2 -7964.59} C_VEL
LIN {X 0,Y 460.473,Z 152.622,A -85,B 0,C 180,E1 -7967.813,E2 -7967.813} C_VEL
LIN {X 0,Y 460.475,Z 152.623,A -85,B 0,C 180,E1 -7970.131,E2 -7970.131} C_VEL
LIN {X 0,Y 460.473,Z 152.629,A -85,B 0,C 180,E1 -7972.529,E2 -7972.529} C_VEL
LIN {X 0,Y 460.485,Z 152.62,A -85,B 0,C 180,E1 -7975.618,E2 -7975.618} C_VEL
LIN {X 0,Y 460.508,Z 152.624,A -85,B 0,C 180,E1 -7978.742,E2 -7978.742} C_VEL
LIN {X 0,Y 460.498,Z 152.624,A -85,B 0,C 180,E1 -7981.763,E2 -7981.763} C_VEL
LIN {X 0,Y 460.57,Z 152.817,A -85,B 0,C 180,E1 -7984.826,E2 -7984.826} C_VEL
LIN {X 0,Y 462.691,Z 164.337,A -85,B 0,C 180,E1 -7987.211,E2 -7987.211} C_VEL
LIN {X 0,Y 462.09,Z 176.505,A -85,B 0,C 180,E1 -7989.524,E2 -7989.524} C_VEL
LIN {X 0,Y 461.485,Z 191.085,A -85,B 0,C 180,E1 -7992.266,E2 -7992.266} C_VEL
LIN {X 0,Y 461.441,Z 193.988,A -85,B 0,C 180,E1 -7992.747,E2 -7992.747} C_VEL
LIN {X 0,Y 464.379,Z 212.326,A -85,B 0,C 180,E1 -7993.174,E2 -7993.174} C_VEL
LIN {X 0,Y 463.609,Z 301.797,A -85,B 0,C 180,E1 -7994.615,E2 -7994.615} C_VEL
LIN {X 0,Y 463.191,Z 315.677,A -85,B 0,C 180,E1 -7995.023,E2 -7995.023} C_VEL
LIN {X 0,Y 462.71,Z 328.658,A -85,B 0,C 180,E1 -7995.598,E2 -7995.598} C_VEL
LIN {X 0,Y 462.22,Z 341.25,A -85,B 0,C 180,E1 -7996.368,E2 -7996.368} C_VEL
LIN {X 0,Y 461.699,Z 352.195,A -85,B 0,C 180,E1 -7997.223,E2 -7997.223} C_VEL
LIN {X 0,Y 461.255,Z 361.567,A -85,B 0,C 180,E1 -7998.129,E2 -7998.129} C_VEL
LIN {X 0,Y 460.753,Z 370.886,A -85,B 0,C 180,E1 -7999.23,E2 -7999.23} C_VEL
LIN {X 0,Y 460.298,Z 379.92,A -85,B 0,C 180,E1 -8000.552,E2 -8000.552} C_VEL
LIN {X 0,Y 459.999,Z 387.195,A -85,B 0,C 180,E1 -8001.875,E2 -8001.875} C_VEL
LIN {X 0,Y 459.747,Z 393.293,A -85,B 0,C 180,E1 -8003.272,E2 -8003.272} C_VEL
LIN {X 0,Y 459.682,Z 398.203,A -85,B 0,C 180,E1 -8004.736,E2 -8004.736} C_VEL
LIN {X 0,Y 459.565,Z 400.515,A -85,B 0,C 180,E1 -8005.614,E2 -8005.614} C_VEL
LIN {X 0,Y 459.558,Z 402.397,A -85,B 0,C 180,E1 -8006.492,E2 -8006.492} C_VEL
LIN {X 0,Y 459.567,Z 403.811,A -85,B 0,C 180,E1 -8007.37,E2 -8007.37} C_VEL
LIN {X 0,Y 459.495,Z 405.429,A -85,B 0,C 180,E1 -8009.123,E2 -8009.123} C_VEL
LIN {X 0,Y 459.502,Z 405.653,A -85,B 0,C 180,E1 -8009.999,E2 -8009.999} C_VEL
LIN {X 0,Y 459.495,Z 405.441,A -85,B 0,C 180,E1 -8010.875,E2 -8010.875} C_VEL
LIN {X 0,Y 459.567,Z 403.835,A -85,B 0,C 180,E1 -8012.629,E2 -8012.629} C_VEL
LIN {X 0,Y 459.557,Z 402.435,A -85,B 0,C 180,E1 -8013.506,E2 -8013.506} C_VEL
LIN {X 0,Y 459.623,Z 399.49,A -85,B 0,C 180,E1 -8014.823,E2 -8014.823} C_VEL
LIN {X 0,Y 459.698,Z 395.503,A -85,B 0,C 180,E1 -8016.142,E2 -8016.142} C_VEL
LIN {X 0,Y 459.905,Z 389.371,A -85,B 0,C 180,E1 -8017.683,E2 -8017.683} C_VEL
LIN {X 0,Y 460.188,Z 382.669,A -85,B 0,C 180,E1 -8019.005,E2 -8019.005} C_VEL
LIN {X 0,Y 460.57,Z 374.354,A -85,B 0,C 180,E1 -8020.328,E2 -8020.328} C_VEL
LIN {X 0,Y 461.076,Z 365.822,A -85,B 0,C 180,E1 -8021.428,E2 -8021.428} C_VEL
LIN {X 0,Y 461.594,Z 355.727,A -85,B 0,C 180,E1 -8022.487,E2 -8022.487} C_VEL
LIN {X 0,Y 462.064,Z 344.852,A -85,B 0,C 180,E1 -8023.411,E2 -8023.411} C_VEL
LIN {X 0,Y 462.571,Z 333.416,A -85,B 0,C 180,E1 -8024.18,E2 -8024.18} C_VEL
LIN {X 0,Y 463.113,Z 321.621,A -85,B 0,C 180,E1 -8024.781,E2 -8024.781} C_VEL
LIN {X 0,Y 463.518,Z 308.061,A -85,B 0,C 180,E1 -8025.273,E2 -8025.273} C_VEL
LIN {X 0,Y 463.812,Z 294.407,A -85,B 0,C 180,E1 -8025.573,E2 -8025.573} C_VEL
LIN {X 0,Y 464.394,Z 211.294,A -85,B 0,C 180,E1 -8026.907,E2 -8026.907} C_VEL
LIN {X 0,Y 461.467,Z 193.635,A -85,B 0,C 180,E1 -8027.336,E2 -8027.336} C_VEL
LIN {X 0,Y 461.812,Z 184.335,A -85,B 0,C 180,E1 -8029.004,E2 -8029.004} C_VEL
LIN {X 0,Y 462.669,Z 165.425,A -85,B 0,C 180,E1 -8032.552,E2 -8032.552} C_VEL
LIN {X 0,Y 461.97,Z 159.922,A -85,B 0,C 180,E1 -8033.648,E2 -8033.648} C_VEL
LIN {X 0,Y 460.573,Z 152.744,A -85,B 0,C 180,E1 -8035.172,E2 -8035.172} C_VEL
LIN {X 0,Y 460.493,Z 152.625,A -85,B 0,C 180,E1 -8038.235,E2 -8038.235} C_VEL
LIN {X 0,Y 460.491,Z 152.624,A -85,B 0,C 180,E1 -8041.276,E2 -8041.276} C_VEL
LIN {X 0,Y 460.514,Z 152.62,A -85,B 0,C 180,E1 -8044.502,E2 -8044.502} C_VEL
LIN {X 0,Y 460.475,Z 152.628,A -85,B 0,C 180,E1 -8047.624,E2 -8047.624} C_VEL
LIN {X 0,Y 460.507,Z 152.622,A -85,B 0,C 180,E1 -8051.012,E2 -8051.012} C_VEL
LIN {X 0,Y 460.502,Z 152.619,A -85,B 0,C 180,E1 -8054.588,E2 -8054.588} C_VEL
LIN {X 0,Y 460.465,Z 152.627,A -85,B 0,C 180,E1 -8057.812,E2 -8057.812} C_VEL
LIN {X 0,Y 460.501,Z 152.619,A -85,B 0,C 180,E1 -8060.134,E2 -8060.134} C_VEL
LIN {X 0,Y 460.456,Z 152.63,A -85,B 0,C 180,E1 -8063.468,E2 -8063.468} C_VEL
LIN {X 0,Y 460.505,Z 152.62,A -85,B 0,C 180,E1 -8066.673,E2 -8066.673} C_VEL
LIN {X 0,Y 460.482,Z 152.622,A -85,B 0,C 180,E1 -8069.757,E2 -8069.757} C_VEL
LIN {X 0,Y 460.478,Z 152.624,A -85,B 0,C 180,E1 -8072.75,E2 -8072.75} C_VEL
LIN {X 0,Y 460.504,Z 152.618,A -85,B 0,C 180,E1 -8075.665,E2 -8075.665} C_VEL
LIN {X 0,Y 460.509,Z 152.621,A -85,B 0,C 180,E1 -8078.577,E2 -8078.577} C_VEL
LIN {X 0,Y 460.571,Z 152.612,A -85,B 0,C 180,E1 -8081.31,E2 -8081.31} C_VEL
LIN {X 0,Y 460.592,Z 152.607,A -85,B 0,C 180,E1 -8084.058,E2 -8084.058} C_VEL
LIN {X 0,Y 460.596,Z 152.607,A -85,B 0,C 180,E1 -8087.665,E2 -8087.665} C_VEL
LIN {X 0,Y 460.603,Z 152.608,A -85,B 0,C 180,E1 -8091.223,E2 -8091.223} C_VEL
LIN {X 0,Y 460.675,Z 152.597,A -85,B 0,C 180,E1 -8093.869,E2 -8093.869} C_VEL
LIN {X 0,Y 460.752,Z 152.588,A -85,B 0,C 180,E1 -8097.377,E2 -8097.377} C_VEL
LIN {X 0,Y 460.781,Z 152.584,A -85,B 0,C 180,E1 -8100,E2 -8100} C_VEL
LIN {X 0,Y 460.747,Z 152.592,A -85,B 0,C 180,E1 -8102.622,E2 -8102.622} C_VEL
LIN {X 0,Y 460.673,Z 152.602,A -85,B 0,C 180,E1 -8106.13,E2 -8106.13} C_VEL
LIN {X 0,Y 460.592,Z 152.61,A -85,B 0,C 180,E1 -8108.776,E2 -8108.776} C_VEL
LIN {X 0,Y 460.582,Z 152.616,A -85,B 0,C 180,E1 -8112.435,E2 -8112.435} C_VEL
LIN {X 0,Y 460.587,Z 152.614,A -85,B 0,C 180,E1 -8115.998,E2 -8115.998} C_VEL
LIN {X 0,Y 460.552,Z 152.615,A -85,B 0,C 180,E1 -8119.616,E2 -8119.616} C_VEL
LIN {X 0,Y 460.496,Z 152.626,A -85,B 0,C 180,E1 -8122.429,E2 -8122.429} C_VEL
LIN {X 0,Y 460.518,Z 152.621,A -85,B 0,C 180,E1 -8125.793,E2 -8125.793} C_VEL
LIN {X 0,Y 460.506,Z 152.624,A -85,B 0,C 180,E1 -8129.233,E2 -8129.233} C_VEL
LIN {X 0,Y 460.57,Z 152.689,A -85,B 0,C 180,E1 -8131.125,E2 -8131.125} C_VEL
LIN {X 0,Y 462.076,Z 161.028,A -85,B 0,C 180,E1 -8132.938,E2 -8132.938} C_VEL
LIN {X 0,Y 461.81,Z 173.112,A -85,B 0,C 180,E1 -8135.33,E2 -8135.33} C_VEL
LIN {X 0,Y 461.553,Z 180.353,A -85,B 0,C 180,E1 -8136.702,E2 -8136.702} C_VEL
LIN {X 0,Y 463.089,Z 188.407,A -85,B 0,C 180,E1 -8136.933,E2 -8136.933} C_VEL
LIN {X 0,Y 464.636,Z 197.605,A -85,B 0,C 180,E1 -8137.146,E2 -8137.146} C_VEL
LIN {X 0,Y 463.717,Z 287.919,A -85,B 0,C 180,E1 -8138.608,E2 -8138.608} C_VEL
LIN {X 0,Y 463.427,Z 301.259,A -85,B 0,C 180,E1 -8139.002,E2 -8139.002} C_VEL
LIN {X 0,Y 462.995,Z 313.923,A -85,B 0,C 180,E1 -8139.556,E2 -8139.556} C_VEL
LIN {X 0,Y 462.504,Z 326.312,A -85,B 0,C 180,E1 -8140.301,E2 -8140.301} C_VEL
LIN {X 0,Y 461.96,Z 337.254,A -85,B 0,C 180,E1 -8141.146,E2 -8141.146} C_VEL
LIN {X 0,Y 461.459,Z 347.678,A -85,B 0,C 180,E1 -8142.149,E2 -8142.149} C_VEL
LIN {X 0,Y 460.911,Z 357.483,A -85,B 0,C 180,E1 -8143.326,E2 -8143.326} C_VEL
LIN {X 0,Y 460.445,Z 366.035,A -85,B 0,C 180,E1 -8144.597,E2 -8144.597} C_VEL
LIN {X 0,Y 460.127,Z 373.02,A -85,B 0,C 180,E1 -8145.879,E2 -8145.879} C_VEL
LIN {X 0,Y 459.908,Z 378.716,A -85,B 0,C 180,E1 -8147.18,E2 -8147.18} C_VEL
LIN {X 0,Y 459.733,Z 383.303,A -85,B 0,C 180,E1 -8148.509,E2 -8148.509} C_VEL
LIN {X 0,Y 459.576,Z 387.206,A -85,B 0,C 180,E1 -8150.04,E2 -8150.04} C_VEL
LIN {X 0,Y 459.437,Z 389.411,A -85,B 0,C 180,E1 -8151.273,E2 -8151.273} C_VEL
LIN {X 0,Y 459.362,Z 390.922,A -85,B 0,C 180,E1 -8152.709,E2 -8152.709} C_VEL
LIN {X 0,Y 459.364,Z 391.352,A -85,B 0,C 180,E1 -8154.18,E2 -8154.18} C_VEL
LIN {X 0,Y 459.405,Z 390.618,A -85,B 0,C 180,E1 -8155.699,E2 -8155.699} C_VEL
LIN {X 0,Y 459.473,Z 388.587,A -85,B 0,C 180,E1 -8157.273,E2 -8157.273} C_VEL
LIN {X 0,Y 459.655,Z 385.097,A -85,B 0,C 180,E1 -8158.894,E2 -8158.894} C_VEL
LIN {X 0,Y 459.75,Z 381.978,A -85,B 0,C 180,E1 -8159.94,E2 -8159.94} C_VEL
LIN {X 0,Y 459.171,Z 379.677,A -85,B 0,C 180,E1 -8160.616,E2 -8160.616} C_VEL
LIN {X 0,Y 456.461,Z 375.525,A -85,B 0,C 180,E1 -8161.693,E2 -8161.693} C_VEL
LIN {X 0,Y 453.806,Z 370.735,A -85,B 0,C 180,E1 -8162.737,E2 -8162.737} C_VEL
LIN {X 0,Y 453.32,Z 367.422,A -85,B 0,C 180,E1 -8163.355,E2 -8163.355} C_VEL
LIN {X 0,Y 453.719,Z 359.903,A -85,B 0,C 180,E1 -8164.544,E2 -8164.544} C_VEL
LIN {X 0,Y 454.244,Z 350.031,A -85,B 0,C 180,E1 -8165.803,E2 -8165.803} C_VEL
LIN {X 0,Y 454.837,Z 339.153,A -85,B 0,C 180,E1 -8166.917,E2 -8166.917} C_VEL
LIN {X 0,Y 455.399,Z 328.092,A -85,B 0,C 180,E1 -8167.812,E2 -8167.812} C_VEL
LIN {X 0,Y 455.923,Z 315.859,A -85,B 0,C 180,E1 -8168.585,E2 -8168.585} C_VEL
LIN {X 0,Y 456.332,Z 304.275,A -85,B 0,C 180,E1 -8169.137,E2 -8169.137} C_VEL
LIN {X 0,Y 456.663,Z 291.24,A -85,B 0,C 180,E1 -8169.569,E2 -8169.569} C_VEL
LIN {X 0,Y 456.898,Z 272.443,A -85,B 0,C 180,E1 -8169.922,E2 -8169.922} C_VEL
LIN {X 0,Y 457.464,Z 196.761,A -85,B 0,C 180,E1 -8171.146,E2 -8171.146} C_VEL
LIN {X 0,Y 454.54,Z 180.637,A -85,B 0,C 180,E1 -8171.551,E2 -8171.551} C_VEL
LIN {X 0,Y 454.666,Z 177.063,A -85,B 0,C 180,E1 -8172.226,E2 -8172.226} C_VEL
LIN {X 0,Y 455.241,Z 162.624,A -85,B 0,C 180,E1 -8175.244,E2 -8175.244} C_VEL
LIN {X 0,Y 453.566,Z 153.544,A -85,B 0,C 180,E1 -8177.33,E2 -8177.33} C_VEL
LIN {X 0,Y 453.589,Z 153.481,A -85,B 0,C 180,E1 -8181.088,E2 -8181.088} C_VEL
LIN {X 0,Y 453.674,Z 153.476,A -85,B 0,C 180,E1 -8183.776,E2 -8183.776} C_VEL
LIN {X 0,Y 453.741,Z 153.463,A -85,B 0,C 180,E1 -8187.338,E2 -8187.338} C_VEL
LIN {X 0,Y 453.82,Z 153.455,A -85,B 0,C 180,E1 -8190.001,E2 -8190.001} C_VEL
LIN {X 0,Y 453.741,Z 153.461,A -85,B 0,C 180,E1 -8192.664,E2 -8192.664} C_VEL
LIN {X 0,Y 453.664,Z 153.471,A -85,B 0,C 180,E1 -8196.226,E2 -8196.226} C_VEL
LIN {X 0,Y 453.584,Z 153.481,A -85,B 0,C 180,E1 -8198.914,E2 -8198.914} C_VEL
LIN {X 0,Y 453.562,Z 153.483,A -85,B 0,C 180,E1 -8202.53,E2 -8202.53} C_VEL
LIN {X 0,Y 453.543,Z 153.486,A -85,B 0,C 180,E1 -8206.197,E2 -8206.197} C_VEL
LIN {X 0,Y 453.516,Z 153.493,A -85,B 0,C 180,E1 -8209.04,E2 -8209.04} C_VEL
LIN {X 0,Y 453.475,Z 153.495,A -85,B 0,C 180,E1 -8211.837,E2 -8211.837} C_VEL
LIN {X 0,Y 453.499,Z 153.493,A -85,B 0,C 180,E1 -8214.736,E2 -8214.736} C_VEL
LIN {X 0,Y 453.531,Z 153.487,A -85,B 0,C 180,E1 -8217.96,E2 -8217.96} C_VEL
LIN {X 0,Y 453.464,Z 153.497,A -85,B 0,C 180,E1 -8221.525,E2 -8221.525} C_VEL
LIN {X 0,Y 453.481,Z 153.498,A -85,B 0,C 180,E1 -8224.777,E2 -8224.777} C_VEL
LIN {X 0,Y 453.461,Z 153.497,A -85,B 0,C 180,E1 -8228.312,E2 -8228.312} C_VEL
LIN {X 0,Y 453.493,Z 153.496,A -85,B 0,C 180,E1 -8230.61,E2 -8230.61} C_VEL
LIN {X 0,Y 453.454,Z 153.499,A -85,B 0,C 180,E1 -8233.245,E2 -8233.245} C_VEL
LIN {X 0,Y 453.459,Z 153.496,A -85,B 0,C 180,E1 -8235.779,E2 -8235.779} C_VEL
LIN {X 0,Y 453.493,Z 153.492,A -85,B 0,C 180,E1 -8239.41,E2 -8239.41} C_VEL
LIN {X 0,Y 453.448,Z 153.502,A -85,B 0,C 180,E1 -8242.81,E2 -8242.81} C_VEL
LIN {X 0,Y 453.475,Z 153.496,A -85,B 0,C 180,E1 -8246.088,E2 -8246.088} C_VEL
LIN {X 0,Y 453.474,Z 153.494,A -85,B 0,C 180,E1 -8249.241,E2 -8249.241} C_VEL
LIN {X 0,Y 453.507,Z 153.497,A -85,B 0,C 180,E1 -8252.296,E2 -8252.296} C_VEL
LIN {X 0,Y 453.494,Z 153.491,A -85,B 0,C 180,E1 -8255.265,E2 -8255.265} C_VEL
LIN {X 0,Y 453.48,Z 153.499,A -85,B 0,C 180,E1 -8258.416,E2 -8258.416} C_VEL
LIN {X 0,Y 453.522,Z 153.488,A -85,B 0,C 180,E1 -8261.009,E2 -8261.009} C_VEL
LIN {X 0,Y 453.569,Z 153.487,A -85,B 0,C 180,E1 -8263.88,E2 -8263.88} C_VEL
LIN {X 0,Y 453.564,Z 153.484,A -85,B 0,C 180,E1 -8267.472,E2 -8267.472} C_VEL
LIN {X 0,Y 453.577,Z 153.481,A -85,B 0,C 180,E1 -8271.087,E2 -8271.087} C_VEL
LIN {X 0,Y 453.636,Z 153.48,A -85,B 0,C 180,E1 -8273.775,E2 -8273.775} C_VEL
LIN {X 0,Y 453.704,Z 153.467,A -85,B 0,C 180,E1 -8277.337,E2 -8277.337} C_VEL
LIN {X 0,Y 453.767,Z 153.462,A -85,B 0,C 180,E1 -8280,E2 -8280} C_VEL
LIN {X 0,Y 453.714,Z 153.464,A -85,B 0,C 180,E1 -8282.664,E2 -8282.664} C_VEL
LIN {X 0,Y 453.628,Z 153.476,A -85,B 0,C 180,E1 -8286.226,E2 -8286.226} C_VEL
LIN {X 0,Y 453.561,Z 153.484,A -85,B 0,C 180,E1 -8288.914,E2 -8288.914} C_VEL
LIN {X 0,Y 453.566,Z 153.482,A -85,B 0,C 180,E1 -8292.529,E2 -8292.529} C_VEL
LIN {X 0,Y 453.538,Z 153.486,A -85,B 0,C 180,E1 -8296.197,E2 -8296.197} C_VEL
LIN {X 0,Y 453.518,Z 153.492,A -85,B 0,C 180,E1 -8299.039,E2 -8299.039} C_VEL
LIN {X 0,Y 453.476,Z 153.495,A -85,B 0,C 180,E1 -8301.837,E2 -8301.837} C_VEL
LIN {X 0,Y 453.463,Z 153.497,A -85,B 0,C 180,E1 -8304.738,E2 -8304.738} C_VEL
LIN {X 0,Y 453.457,Z 153.496,A -85,B 0,C 180,E1 -8307.941,E2 -8307.941} C_VEL
LIN {X 0,Y 453.448,Z 153.501,A -85,B 0,C 180,E1 -8310.762,E2 -8310.762} C_VEL
LIN {X 0,Y 453.456,Z 153.496,A -85,B 0,C 180,E1 -8313.915,E2 -8313.915} C_VEL
LIN {X 0,Y 453.436,Z 153.504,A -85,B 0,C 180,E1 -8317.192,E2 -8317.192} C_VEL
LIN {X 0,Y 453.466,Z 153.499,A -85,B 0,C 180,E1 -8320.612,E2 -8320.612} C_VEL
LIN {X 0,Y 453.483,Z 153.497,A -85,B 0,C 180,E1 -8324.528,E2 -8324.528} C_VEL
LIN {X 0,Y 453.433,Z 153.5,A -85,B 0,C 180,E1 -8328.072,E2 -8328.072} C_VEL
LIN {X 0,Y 453.424,Z 153.506,A -85,B 0,C 180,E1 -8330.805,E2 -8330.805} C_VEL
LIN {X 0,Y 453.407,Z 153.503,A -85,B 0,C 180,E1 -8333.912,E2 -8333.912} C_VEL
LIN {X 0,Y 453.439,Z 153.499,A -85,B 0,C 180,E1 -8337.147,E2 -8337.147} C_VEL
LIN {X 0,Y 453.45,Z 153.504,A -85,B 0,C 180,E1 -8340.266,E2 -8340.266} C_VEL
LIN {X 0,Y 453.426,Z 153.502,A -85,B 0,C 180,E1 -8343.288,E2 -8343.288} C_VEL
LIN {X 0,Y 453.502,Z 153.618,A -85,B 0,C 180,E1 -8344.59,E2 -8344.59} C_VEL
LIN {X 0,Y 455.717,Z 165.397,A -85,B 0,C 180,E1 -8347.082,E2 -8347.082} C_VEL
LIN {X 0,Y 455.174,Z 176.349,A -85,B 0,C 180,E1 -8349.198,E2 -8349.198} C_VEL
LIN {X 0,Y 454.51,Z 190.913,A -85,B 0,C 180,E1 -8351.985,E2 -8351.985} C_VEL
LIN {X 0,Y 454.468,Z 193.76,A -85,B 0,C 180,E1 -8352.476,E2 -8352.476} C_VEL
LIN {X 0,Y 456.237,Z 204.889,A -85,B 0,C 180,E1 -8352.76,E2 -8352.76} C_VEL
LIN {X 0,Y 457.553,Z 214.577,A -85,B 0,C 180,E1 -8352.968,E2 -8352.968} C_VEL
LIN {X 0,Y 456.724,Z 302.342,A -85,B 0,C 180,E1 -8354.406,E2 -8354.406} C_VEL
LIN {X 0,Y 456.301,Z 316.003,A -85,B 0,C 180,E1 -8354.82,E2 -8354.82} C_VEL
LIN {X 0,Y 455.839,Z 328.331,A -85,B 0,C 180,E1 -8355.376,E2 -8355.376} C_VEL
LIN {X 0,Y 455.344,Z 339.384,A -85,B 0,C 180,E1 -8356.044,E2 -8356.044} C_VEL
LIN {X 0,Y 454.772,Z 351.283,A -85,B 0,C 180,E1 -8356.967,E2 -8356.967} C_VEL
LIN {X 0,Y 454.3,Z 361.345,A -85,B 0,C 180,E1 -8357.945,E2 -8357.945} C_VEL
LIN {X 0,Y 453.727,Z 370.691,A -85,B 0,C 180,E1 -8359.061,E2 -8359.061} C_VEL
LIN {X 0,Y 453.255,Z 379.741,A -85,B 0,C 180,E1 -8360.404,E2 -8360.404} C_VEL
LIN {X 0,Y 452.931,Z 387.03,A -85,B 0,C 180,E1 -8361.747,E2 -8361.747} C_VEL
LIN {X 0,Y 452.72,Z 391.952,A -85,B 0,C 180,E1 -8362.865,E2 -8362.865} C_VEL
LIN {X 0,Y 452.589,Z 396.731,A -85,B 0,C 180,E1 -8364.206,E2 -8364.206} C_VEL
LIN {X 0,Y 452.488,Z 400.384,A -85,B 0,C 180,E1 -8365.545,E2 -8365.545} C_VEL
LIN {X 0,Y 452.456,Z 402.271,A -85,B 0,C 180,E1 -8366.437,E2 -8366.437} C_VEL
LIN {X 0,Y 452.491,Z 403.691,A -85,B 0,C 180,E1 -8367.328,E2 -8367.328} C_VEL
LIN {X 0,Y 452.404,Z 405.315,A -85,B 0,C 180,E1 -8369.109,E2 -8369.109} C_VEL
LIN {X 0,Y 452.408,Z 405.542,A -85,B 0,C 180,E1 -8369.999,E2 -8369.999} C_VEL
LIN {X 0,Y 452.404,Z 405.334,A -85,B 0,C 180,E1 -8370.889,E2 -8370.889} C_VEL
LIN {X 0,Y 452.491,Z 403.732,A -85,B 0,C 180,E1 -8372.67,E2 -8372.67} C_VEL
LIN {X 0,Y 452.455,Z 402.334,A -85,B 0,C 180,E1 -8373.561,E2 -8373.561} C_VEL
LIN {X 0,Y 452.555,Z 399.392,A -85,B 0,C 180,E1 -8374.899,E2 -8374.899} C_VEL
LIN {X 0,Y 452.629,Z 394.796,A -85,B 0,C 180,E1 -8376.415,E2 -8376.415} C_VEL
LIN {X 0,Y 452.858,Z 389.279,A -85,B 0,C 180,E1 -8377.803,E2 -8377.803} C_VEL
LIN {X 0,Y 453.135,Z 382.58,A -85,B 0,C 180,E1 -8379.146,E2 -8379.146} C_VEL
LIN {X 0,Y 453.559,Z 374.275,A -85,B 0,C 180,E1 -8380.489,E2 -8380.489} C_VEL
LIN {X 0,Y 454.109,Z 365.757,A -85,B 0,C 180,E1 -8381.606,E2 -8381.606} C_VEL
LIN {X 0,Y 454.645,Z 355.898,A -85,B 0,C 180,E1 -8382.66,E2 -8382.66} C_VEL
LIN {X 0,Y 455.146,Z 344.828,A -85,B 0,C 180,E1 -8383.619,E2 -8383.619} C_VEL
LIN {X 0,Y 455.676,Z 333.418,A -85,B 0,C 180,E1 -8384.399,E2 -8384.399} C_VEL
LIN {X 0,Y 456.271,Z 321.673,A -85,B 0,C 180,E1 -8385.007,E2 -8385.007} C_VEL
LIN {X 0,Y 456.67,Z 308.186,A -85,B 0,C 180,E1 -8385.508,E2 -8385.508} C_VEL
LIN {X 0,Y 456.991,Z 294.772,A -85,B 0,C 180,E1 -8385.812,E2 -8385.812} C_VEL
LIN {X 0,Y 457.673,Z 212.431,A -85,B 0,C 180,E1 -8387.152,E2 -8387.152} C_VEL
LIN {X 0,Y 454.53,Z 193.443,A -85,B 0,C 180,E1 -8387.629,E2 -8387.629} C_VEL
LIN {X 0,Y 455.134,Z 178.885,A -85,B 0,C 180,E1 -8390.329,E2 -8390.329} C_VEL
LIN {X 0,Y 455.748,Z 166.602,A -85,B 0,C 180,E1 -8392.675,E2 -8392.675} C_VEL
LIN {X 0,Y 454.631,Z 159.095,A -85,B 0,C 180,E1 -8394.207,E2 -8394.207} C_VEL
LIN {X 0,Y 453.507,Z 153.626,A -85,B 0,C 180,E1 -8395.407,E2 -8395.407} C_VEL
LIN {X 0,Y 453.444,Z 153.502,A -85,B 0,C 180,E1 -8398.715,E2 -8398.715} C_VEL
LIN {X 0,Y 453.439,Z 153.506,A -85,B 0,C 180,E1 -8401.8,E2 -8401.8} C_VEL
LIN {X 0,Y 453.466,Z 153.5,A -85,B 0,C 180,E1 -8404.989,E2 -8404.989} C_VEL
LIN {X 0,Y 453.436,Z 153.5,A -85,B 0,C 180,E1 -8408.313,E2 -8408.313} C_VEL
LIN {X 0,Y 453.463,Z 153.497,A -85,B 0,C 180,E1 -8410.61,E2 -8410.61} C_VEL
LIN {X 0,Y 453.472,Z 153.495,A -85,B 0,C 180,E1 -8414.527,E2 -8414.527} C_VEL
LIN {X 0,Y 453.427,Z 153.502,A -85,B 0,C 180,E1 -8418.07,E2 -8418.07} C_VEL
LIN {X 0,Y 453.433,Z 153.503,A -85,B 0,C 180,E1 -8420.8,E2 -8420.8} C_VEL
LIN {X 0,Y 453.438,Z 153.5,A -85,B 0,C 180,E1 -8423.915,E2 -8423.915} C_VEL
LIN {X 0,Y 453.461,Z 153.503,A -85,B 0,C 180,E1 -8427.149,E2 -8427.149} C_VEL
LIN {X 0,Y 453.443,Z 153.498,A -85,B 0,C 180,E1 -8430.266,E2 -8430.266} C_VEL
LIN {X 0,Y 453.428,Z 153.504,A -85,B 0,C 180,E1 -8433.289,E2 -8433.289} C_VEL
LIN {X 0,Y 453.48,Z 153.493,A -85,B 0,C 180,E1 -8436.237,E2 -8436.237} C_VEL
LIN {X 0,Y 453.469,Z 153.499,A -85,B 0,C 180,E1 -8439.117,E2 -8439.117} C_VEL
LIN {X 0,Y 453.487,Z 153.491,A -85,B 0,C 180,E1 -8441.943,E2 -8441.943} C_VEL
LIN {X 0,Y 453.521,Z 153.49,A -85,B 0,C 180,E1 -8444.725,E2 -8444.725} C_VEL
LIN {X 0,Y 453.543,Z 153.488,A -85,B 0,C 180,E1 -8448.378,E2 -8448.378} C_VEL
LIN {X 0,Y 453.569,Z 153.486,A -85,B 0,C 180,E1 -8451.086,E2 -8451.086} C_VEL
LIN {X 0,Y 453.643,Z 153.472,A -85,B 0,C 180,E1 -8453.774,E2 -8453.774} C_VEL
LIN {X 0,Y 453.699,Z 153.467,A -85,B 0,C 180,E1 -8457.336,E2 -8457.336} C_VEL
LIN {X 0,Y 453.732,Z 153.462,A -85,B 0,C 180,E1 -8460,E2 -8460} C_VEL
LIN {X 0,Y 453.694,Z 153.47,A -85,B 0,C 180,E1 -8462.663,E2 -8462.663} C_VEL
LIN {X 0,Y 453.64,Z 153.478,A -85,B 0,C 180,E1 -8466.225,E2 -8466.225} C_VEL
LIN {X 0,Y 453.557,Z 153.485,A -85,B 0,C 180,E1 -8468.914,E2 -8468.914} C_VEL
LIN {X 0,Y 453.55,Z 153.492,A -85,B 0,C 180,E1 -8472.529,E2 -8472.529} C_VEL
LIN {X 0,Y 453.53,Z 153.493,A -85,B 0,C 180,E1 -8476.196,E2 -8476.196} C_VEL
LIN {X 0,Y 453.502,Z 153.493,A -85,B 0,C 180,E1 -8479.039,E2 -8479.039} C_VEL
LIN {X 0,Y 453.462,Z 153.501,A -85,B 0,C 180,E1 -8481.836,E2 -8481.836} C_VEL
LIN {X 0,Y 453.453,Z 153.498,A -85,B 0,C 180,E1 -8484.737,E2 -8484.737} C_VEL
LIN {X 0,Y 453.447,Z 153.504,A -85,B 0,C 180,E1 -8487.943,E2 -8487.943} C_VEL
LIN {X 0,Y 453.501,Z 153.533,A -85,B 0,C 180,E1 -8490.881,E2 -8490.881} C_VEL
LIN {X 0,Y 454.474,Z 158.312,A -85,B 0,C 180,E1 -8491.981,E2 -8491.981} C_VEL
LIN {X 0,Y 455.255,Z 163.624,A -85,B 0,C 180,E1 -8493.104,E2 -8493.104} C_VEL
LIN {X 0,Y 454.638,Z 179.072,A -85,B 0,C 180,E1 -8496.185,E2 -8496.185} C_VEL
LIN {X 0,Y 454.656,Z 180.776,A -85,B 0,C 180,E1 -8496.438,E2 -8496.438} C_VEL
LIN {X 0,Y 457.8,Z 197.554,A -85,B 0,C 180,E1 -8496.872,E2 -8496.872} C_VEL
LIN {X 0,Y 456.872,Z 288.695,A -85,B 0,C 180,E1 -8498.38,E2 -8498.38} C_VEL
LIN {X 0,Y 456.563,Z 302.261,A -85,B 0,C 180,E1 -8498.797,E2 -8498.797} C_VEL
LIN {X 0,Y 456.127,Z 314.874,A -85,B 0,C 180,E1 -8499.371,E2 -8499.371} C_VEL
LIN {X 0,Y 455.656,Z 325.815,A -85,B 0,C 180,E1 -8500.039,E2 -8500.039} C_VEL
LIN {X 0,Y 455.046,Z 337.431,A -85,B 0,C 180,E1 -8500.945,E2 -8500.945} C_VEL
LIN {X 0,Y 454.53,Z 346.942,A -85,B 0,C 180,E1 -8501.867,E2 -8501.867} C_VEL
LIN {X 0,Y 454.038,Z 355.918,A -85,B 0,C 180,E1 -8502.927,E2 -8502.927} C_VEL
LIN {X 0,Y 453.512,Z 364.765,A -85,B 0,C 180,E1 -8504.215,E2 -8504.215} C_VEL
LIN {X 0,Y 453.121,Z 371.996,A -85,B 0,C 180,E1 -8505.517,E2 -8505.517} C_VEL
LIN {X 0,Y 452.852,Z 378.298,A -85,B 0,C 180,E1 -8506.935,E2 -8506.935} C_VEL
LIN {X 0,Y 452.69,Z 382.655,A -85,B 0,C 180,E1 -8508.175,E2 -8508.175} C_VEL
LIN {X 0,Y 452.552,Z 386.384,A -85,B 0,C 180,E1 -8509.548,E2 -8509.548} C_VEL
LIN {X 0,Y 452.38,Z 389.124,A -85,B 0,C 180,E1 -8510.966,E2 -8510.966} C_VEL
LIN {X 0,Y 452.274,Z 391.043,A -85,B 0,C 180,E1 -8512.699,E2 -8512.699} C_VEL
LIN {X 0,Y 452.251,Z 391.472,A -85,B 0,C 180,E1 -8513.908,E2 -8513.908} C_VEL
LIN {X 0,Y 452.314,Z 390.972,A -85,B 0,C 180,E1 -8515.437,E2 -8515.437} C_VEL
LIN {X 0,Y 452.355,Z 389.114,A -85,B 0,C 180,E1 -8517.061,E2 -8517.061} C_VEL
LIN {X 0,Y 452.559,Z 385.93,A -85,B 0,C 180,E1 -8518.662,E2 -8518.662} C_VEL
LIN {X 0,Y 452.712,Z 381.471,A -85,B 0,C 180,E1 -8520.215,E2 -8520.215} C_VEL
LIN {X 0,Y 452.937,Z 375.579,A -85,B 0,C 180,E1 -8521.737,E2 -8521.737} C_VEL
LIN {X 0,Y 453.251,Z 369.227,A -85,B 0,C 180,E1 -8523.03,E2 -8523.03} C_VEL
LIN {X 0,Y 453.32,Z 367.422,A -85,B 0,C 180,E1 -8523.355,E2 -8523.355} C_VEL
LIN {X 0,Y 452.876,Z 363.93,A -85,B 0,C 180,E1 -8523.956,E2 -8523.956} C_VEL
LIN {X 0,Y 450.418,Z 357.969,A -85,B 0,C 180,E1 -8524.912,E2 -8524.912} C_VEL
LIN {X 0,Y 447.945,Z 351.446,A -85,B 0,C 180,E1 -8525.813,E2 -8525.813} C_VEL
LIN {X 0,Y 447.477,Z 347.071,A -85,B 0,C 180,E1 -8526.319,E2 -8526.319} C_VEL
LIN {X 0,Y 448.044,Z 336.659,A -85,B 0,C 180,E1 -8527.333,E2 -8527.333} C_VEL
LIN {X 0,Y 448.607,Z 326.145,A -85,B 0,C 180,E1 -8528.158,E2 -8528.158} C_VEL
LIN {X 0,Y 449.112,Z 313.997,A -85,B 0,C 180,E1 -8528.906,E2 -8528.906} C_VEL
LIN {X 0,Y 449.503,Z 300.772,A -85,B 0,C 180,E1 -8529.498,E2 -8529.498} C_VEL
LIN {X 0,Y 449.887,Z 287.919,A -85,B 0,C 180,E1 -8529.881,E2 -8529.881} C_VEL
LIN {X 0,Y 450.658,Z 197.728,A -85,B 0,C 180,E1 -8531.386,E2 -8531.386} C_VEL
LIN {X 0,Y 447.604,Z 180.808,A -85,B 0,C 180,E1 -8531.818,E2 -8531.818} C_VEL
LIN {X 0,Y 447.694,Z 177.613,A -85,B 0,C 180,E1 -8532.412,E2 -8532.412} C_VEL
LIN {X 0,Y 448.296,Z 164.252,A -85,B 0,C 180,E1 -8535.242,E2 -8535.242} C_VEL
LIN {X 0,Y 446.519,Z 154.432,A -85,B 0,C 180,E1 -8537.521,E2 -8537.521} C_VEL
LIN {X 0,Y 446.535,Z 154.36,A -85,B 0,C 180,E1 -8540.946,E2 -8540.946} C_VEL
LIN {X 0,Y 446.643,Z 154.35,A -85,B 0,C 180,E1 -8543.677,E2 -8543.677} C_VEL
LIN {X 0,Y 446.688,Z 154.341,A -85,B 0,C 180,E1 -8547.296,E2 -8547.296} C_VEL
LIN {X 0,Y 446.79,Z 154.331,A -85,B 0,C 180,E1 -8550.001,E2 -8550.001} C_VEL
LIN {X 0,Y 446.689,Z 154.339,A -85,B 0,C 180,E1 -8552.706,E2 -8552.706} C_VEL
LIN {X 0,Y 446.633,Z 154.347,A -85,B 0,C 180,E1 -8556.325,E2 -8556.325} C_VEL
LIN {X 0,Y 446.532,Z 154.361,A -85,B 0,C 180,E1 -8559.056,E2 -8559.056} C_VEL
LIN {X 0,Y 446.52,Z 154.361,A -85,B 0,C 180,E1 -8562.731,E2 -8562.731} C_VEL
LIN {X 0,Y 446.494,Z 154.364,A -85,B 0,C 180,E1 -8566.228,E2 -8566.228} C_VEL
LIN {X 0,Y 446.467,Z 154.374,A -85,B 0,C 180,E1 -8569.304,E2 -8569.304} C_VEL
LIN {X 0,Y 446.417,Z 154.373,A -85,B 0,C 180,E1 -8572.2,E2 -8572.2} C_VEL
LIN {X 0,Y 446.443,Z 154.377,A -85,B 0,C 180,E1 -8575.154,E2 -8575.154} C_VEL
LIN {X 0,Y 446.484,Z 154.365,A -85,B 0,C 180,E1 -8578.179,E2 -8578.179} C_VEL
LIN {X 0,Y 446.417,Z 154.374,A -85,B 0,C 180,E1 -8581.775,E2 -8581.775} C_VEL
LIN {X 0,Y 446.422,Z 154.375,A -85,B 0,C 180,E1 -8584.524,E2 -8584.524} C_VEL
LIN {X 0,Y 446.413,Z 154.374,A -85,B 0,C 180,E1 -8588.08,E2 -8588.08} C_VEL
LIN {X 0,Y 446.426,Z 154.379,A -85,B 0,C 180,E1 -8590.918,E2 -8590.918} C_VEL
LIN {X 0,Y 446.399,Z 154.375,A -85,B 0,C 180,E1 -8593.847,E2 -8593.847} C_VEL
LIN {X 0,Y 446.397,Z 154.379,A -85,B 0,C 180,E1 -8596.404,E2 -8596.404} C_VEL
LIN {X 0,Y 446.422,Z 154.375,A -85,B 0,C 180,E1 -8599.084,E2 -8599.084} C_VEL
LIN {X 0,Y 446.404,Z 154.377,A -85,B 0,C 180,E1 -8602.121,E2 -8602.121} C_VEL
LIN {X 0,Y 446.427,Z 154.372,A -85,B 0,C 180,E1 -8605.477,E2 -8605.477} C_VEL
LIN {X 0,Y 446.415,Z 154.378,A -85,B 0,C 180,E1 -8608.7,E2 -8608.7} C_VEL
LIN {X 0,Y 446.448,Z 154.371,A -85,B 0,C 180,E1 -8611.831,E2 -8611.831} C_VEL
LIN {X 0,Y 446.439,Z 154.372,A -85,B 0,C 180,E1 -8614.847,E2 -8614.847} C_VEL
LIN {X 0,Y 446.448,Z 154.377,A -85,B 0,C 180,E1 -8618.246,E2 -8618.246} C_VEL
LIN {X 0,Y 446.45,Z 154.371,A -85,B 0,C 180,E1 -8621.649,E2 -8621.649} C_VEL
LIN {X 0,Y 446.506,Z 154.365,A -85,B 0,C 180,E1 -8624.48,E2 -8624.48} C_VEL
LIN {X 0,Y 446.516,Z 154.366,A -85,B 0,C 180,E1 -8628.193,E2 -8628.193} C_VEL
LIN {X 0,Y 446.526,Z 154.359,A -85,B 0,C 180,E1 -8630.945,E2 -8630.945} C_VEL
LIN {X 0,Y 446.606,Z 154.354,A -85,B 0,C 180,E1 -8633.676,E2 -8633.676} C_VEL
LIN {X 0,Y 446.653,Z 154.345,A -85,B 0,C 180,E1 -8637.295,E2 -8637.295} C_VEL
LIN {X 0,Y 446.717,Z 154.341,A -85,B 0,C 180,E1 -8640,E2 -8640} C_VEL
LIN {X 0,Y 446.663,Z 154.342,A -85,B 0,C 180,E1 -8642.706,E2 -8642.706} C_VEL
LIN {X 0,Y 446.599,Z 154.351,A -85,B 0,C 180,E1 -8646.325,E2 -8646.325} C_VEL
LIN {X 0,Y 446.512,Z 154.363,A -85,B 0,C 180,E1 -8649.056,E2 -8649.056} C_VEL
LIN {X 0,Y 446.523,Z 154.36,A -85,B 0,C 180,E1 -8652.73,E2 -8652.73} C_VEL
LIN {X 0,Y 446.485,Z 154.365,A -85,B 0,C 180,E1 -8656.46,E2 -8656.46} C_VEL
LIN {X 0,Y 446.469,Z 154.374,A -85,B 0,C 180,E1 -8659.304,E2 -8659.304} C_VEL
LIN {X 0,Y 446.417,Z 154.373,A -85,B 0,C 180,E1 -8662.2,E2 -8662.2} C_VEL
LIN {X 0,Y 446.414,Z 154.38,A -85,B 0,C 180,E1 -8665.155,E2 -8665.155} C_VEL
LIN {X 0,Y 446.417,Z 154.373,A -85,B 0,C 180,E1 -8668.184,E2 -8668.184} C_VEL
LIN {X 0,Y 446.39,Z 154.382,A -85,B 0,C 180,E1 -8671.303,E2 -8671.303} C_VEL
LIN {X 0,Y 446.415,Z 154.375,A -85,B 0,C 180,E1 -8674.525,E2 -8674.525} C_VEL
LIN {X 0,Y 446.391,Z 154.376,A -85,B 0,C 180,E1 -8677.881,E2 -8677.881} C_VEL
LIN {X 0,Y 446.397,Z 154.377,A -85,B 0,C 180,E1 -8681.395,E2 -8681.395} C_VEL
LIN {X 0,Y 446.423,Z 154.376,A -85,B 0,C 180,E1 -8685.108,E2 -8685.108} C_VEL
LIN {X 0,Y 446.397,Z 154.382,A -85,B 0,C 180,E1 -8688.605,E2 -8688.605} C_VEL
LIN {X 0,Y 446.385,Z 154.379,A -85,B 0,C 180,E1 -8692.118,E2 -8692.118} C_VEL
LIN {X 0,Y 446.372,Z 154.379,A -85,B 0,C 180,E1 -8695.471,E2 -8695.471} C_VEL
LIN {X 0,Y 446.39,Z 154.383,A -85,B 0,C 180,E1 -8698.697,E2 -8698.697} C_VEL
LIN {X 0,Y 446.403,Z 154.38,A -85,B 0,C 180,E1 -8701.842,E2 -8701.842} C_VEL
LIN {X 0,Y 446.492,Z 154.569,A -85,B 0,C 180,E1 -8704.412,E2 -8704.412} C_VEL
LIN {X 0,Y 448.749,Z 166.448,A -85,B 0,C 180,E1 -8706.949,E2 -8706.949} C_VEL
LIN {X 0,Y 448.316,Z 176.186,A -85,B 0,C 180,E1 -8708.865,E2 -8708.865} C_VEL
LIN {X 0,Y 447.499,Z 192.068,A -85,B 0,C 180,E1 -8711.952,E2 -8711.952} C_VEL
LIN {X 0,Y 447.494,Z 193.662,A -85,B 0,C 180,E1 -8712.205,E2 -8712.205} C_VEL
LIN {X 0,Y 448.669,Z 200.869,A -85,B 0,C 180,E1 -8712.409,E2 -8712.409} C_VEL
LIN {X 0,Y 450.739,Z 213.982,A -85,B 0,C 180,E1 -8712.708,E2 -8712.708} C_VEL
LIN {X 0,Y 449.903,Z 301.598,A -85,B 0,C 180,E1 -8714.163,E2 -8714.163} C_VEL
LIN {X 0,Y 449.455,Z 315.466,A -85,B 0,C 180,E1 -8714.583,E2 -8714.583} C_VEL
LIN {X 0,Y 448.949,Z 327.928,A -85,B 0,C 180,E1 -8715.146,E2 -8715.146} C_VEL
LIN {X 0,Y 448.424,Z 339.057,A -85,B 0,C 180,E1 -8715.824,E2 -8715.824} C_VEL
LIN {X 0,Y 447.836,Z 351.003,A -85,B 0,C 180,E1 -8716.762,E2 -8716.762} C_VEL
LIN {X 0,Y 447.335,Z 361.1,A -85,B 0,C 180,E1 -8717.754,E2 -8717.754} C_VEL
LIN {X 0,Y 446.724,Z 370.484,A -85,B 0,C 180,E1 -8718.888,E2 -8718.888} C_VEL
LIN {X 0,Y 446.226,Z 379.556,A -85,B 0,C 180,E1 -8720.251,E2 -8720.251} C_VEL
LIN {X 0,Y 445.859,Z 386.862,A -85,B 0,C 180,E1 -8721.615,E2 -8721.615} C_VEL
LIN {X 0,Y 445.667,Z 391.799,A -85,B 0,C 180,E1 -8722.752,E2 -8722.752} C_VEL
LIN {X 0,Y 445.499,Z 395.984,A -85,B 0,C 180,E1 -8723.922,E2 -8723.922} C_VEL
LIN {X 0,Y 445.415,Z 400.252,A -85,B 0,C 180,E1 -8725.474,E2 -8725.474} C_VEL
LIN {X 0,Y 445.355,Z 402.143,A -85,B 0,C 180,E1 -8726.38,E2 -8726.38} C_VEL
LIN {X 0,Y 445.399,Z 403.57,A -85,B 0,C 180,E1 -8727.286,E2 -8727.286} C_VEL
LIN {X 0,Y 445.352,Z 404.58,A -85,B 0,C 180,E1 -8728.19,E2 -8728.19} C_VEL
LIN {X 0,Y 445.317,Z 405.431,A -85,B 0,C 180,E1 -8729.999,E2 -8729.999} C_VEL
LIN {X 0,Y 445.315,Z 405.227,A -85,B 0,C 180,E1 -8730.903,E2 -8730.903} C_VEL
LIN {X 0,Y 445.398,Z 403.63,A -85,B 0,C 180,E1 -8732.712,E2 -8732.712} C_VEL
LIN {X 0,Y 445.355,Z 402.235,A -85,B 0,C 180,E1 -8733.618,E2 -8733.618} C_VEL
LIN {X 0,Y 445.487,Z 399.298,A -85,B 0,C 180,E1 -8734.977,E2 -8734.977} C_VEL
LIN {X 0,Y 445.612,Z 393.888,A -85,B 0,C 180,E1 -8736.747,E2 -8736.747} C_VEL
LIN {X 0,Y 445.84,Z 388.187,A -85,B 0,C 180,E1 -8738.155,E2 -8738.155} C_VEL
LIN {X 0,Y 446.197,Z 381.272,A -85,B 0,C 180,E1 -8739.518,E2 -8739.518} C_VEL
LIN {X 0,Y 446.626,Z 372.622,A -85,B 0,C 180,E1 -8740.883,E2 -8740.883} C_VEL
LIN {X 0,Y 447.289,Z 363.753,A -85,B 0,C 180,E1 -8742.015,E2 -8742.015} C_VEL
LIN {X 0,Y 447.844,Z 353.449,A -85,B 0,C 180,E1 -8743.092,E2 -8743.092} C_VEL
LIN {X 0,Y 448.333,Z 343.375,A -85,B 0,C 180,E1 -8743.945,E2 -8743.945} C_VEL
LIN {X 0,Y 448.913,Z 331.482,A -85,B 0,C 180,E1 -8744.737,E2 -8744.737} C_VEL
LIN {X 0,Y 449.53,Z 319.135,A -85,B 0,C 180,E1 -8745.354,E2 -8745.354} C_VEL
LIN {X 0,Y 449.928,Z 306.495,A -85,B 0,C 180,E1 -8745.805,E2 -8745.805} C_VEL
LIN {X 0,Y 450.226,Z 291.648,A -85,B 0,C 180,E1 -8746.114,E2 -8746.114} C_VEL
LIN {X 0,Y 450.895,Z 213.11,A -85,B 0,C 180,E1 -8747.417,E2 -8747.417} C_VEL
LIN {X 0,Y 447.592,Z 193.487,A -85,B 0,C 180,E1 -8747.919,E2 -8747.919} C_VEL
LIN {X 0,Y 447.613,Z 191.111,A -85,B 0,C 180,E1 -8748.3,E2 -8748.3} C_VEL
LIN {X 0,Y 448.496,Z 173.924,A -85,B 0,C 180,E1 -8751.606,E2 -8751.606} C_VEL
LIN {X 0,Y 448.737,Z 166.561,A -85,B 0,C 180,E1 -8753.049,E2 -8753.049} C_VEL
LIN {X 0,Y 446.932,Z 156.75,A -85,B 0,C 180,E1 -8755.122,E2 -8755.122} C_VEL
LIN {X 0,Y 446.457,Z 154.443,A -85,B 0,C 180,E1 -8755.681,E2 -8755.681} C_VEL
LIN {X 0,Y 446.404,Z 154.38,A -85,B 0,C 180,E1 -8759.211,E2 -8759.211} C_VEL
LIN {X 0,Y 446.404,Z 154.378,A -85,B 0,C 180,E1 -8762.361,E2 -8762.361} C_VEL
LIN {X 0,Y 446.415,Z 154.379,A -85,B 0,C 180,E1 -8765.05,E2 -8765.05} C_VEL
LIN {X 0,Y 446.389,Z 154.379,A -85,B 0,C 180,E1 -8768.074,E2 -8768.074} C_VEL
LIN {X 0,Y 446.393,Z 154.383,A -85,B 0,C 180,E1 -8771.393,E2 -8771.393} C_VEL
LIN {X 0,Y 446.413,Z 154.379,A -85,B 0,C 180,E1 -8775.106,E2 -8775.106} C_VEL
LIN {X 0,Y 446.391,Z 154.379,A -85,B 0,C 180,E1 -8778.604,E2 -8778.604} C_VEL
LIN {X 0,Y 446.392,Z 154.375,A -85,B 0,C 180,E1 -8781.922,E2 -8781.922} C_VEL
LIN {X 0,Y 446.411,Z 154.375,A -85,B 0,C 180,E1 -8785.475,E2 -8785.475} C_VEL
LIN {X 0,Y 446.381,Z 154.381,A -85,B 0,C 180,E1 -8788.697,E2 -8788.697} C_VEL
LIN {X 0,Y 446.413,Z 154.373,A -85,B 0,C 180,E1 -8791.835,E2 -8791.835} C_VEL
LIN {X 0,Y 446.408,Z 154.381,A -85,B 0,C 180,E1 -8794.844,E2 -8794.844} C_VEL
LIN {X 0,Y 446.436,Z 154.371,A -85,B 0,C 180,E1 -8798.244,E2 -8798.244} C_VEL
LIN {X 0,Y 446.437,Z 154.37,A -85,B 0,C 180,E1 -8801.648,E2 -8801.648} C_VEL
LIN {X 0,Y 446.491,Z 154.366,A -85,B 0,C 180,E1 -8804.479,E2 -8804.479} C_VEL
LIN {X 0,Y 446.502,Z 154.364,A -85,B 0,C 180,E1 -8808.192,E2 -8808.192} C_VEL
LIN {X 0,Y 446.516,Z 154.366,A -85,B 0,C 180,E1 -8810.944,E2 -8810.944} C_VEL
LIN {X 0,Y 446.613,Z 154.348,A -85,B 0,C 180,E1 -8813.675,E2 -8813.675} C_VEL
LIN {X 0,Y 446.649,Z 154.345,A -85,B 0,C 180,E1 -8817.294,E2 -8817.294} C_VEL
LIN {X 0,Y 446.683,Z 154.34,A -85,B 0,C 180,E1 -8820,E2 -8820} C_VEL
LIN {X 0,Y 446.643,Z 154.347,A -85,B 0,C 180,E1 -8822.705,E2 -8822.705} C_VEL
LIN {X 0,Y 446.61,Z 154.353,A -85,B 0,C 180,E1 -8826.324,E2 -8826.324} C_VEL
LIN {X 0,Y 446.504,Z 154.363,A -85,B 0,C 180,E1 -8829.056,E2 -8829.056} C_VEL
LIN {X 0,Y 446.507,Z 154.366,A -85,B 0,C 180,E1 -8832.73,E2 -8832.73} C_VEL
LIN {X 0,Y 446.473,Z 154.373,A -85,B 0,C 180,E1 -8836.459,E2 -8836.459} C_VEL
LIN {X 0,Y 446.454,Z 154.371,A -85,B 0,C 180,E1 -8839.303,E2 -8839.303} C_VEL
LIN {X 0,Y 446.404,Z 154.381,A -85,B 0,C 180,E1 -8842.2,E2 -8842.2} C_VEL
LIN {X 0,Y 446.405,Z 154.375,A -85,B 0,C 180,E1 -8845.155,E2 -8845.155} C_VEL
LIN {X 0,Y 446.402,Z 154.381,A -85,B 0,C 180,E1 -8848.184,E2 -8848.184} C_VEL
LIN {X 0,Y 446.502,Z 154.515,A -85,B 0,C 180,E1 -8850.701,E2 -8850.701} C_VEL
LIN {X 0,Y 448.22,Z 163.719,A -85,B 0,C 180,E1 -8852.748,E2 -8852.748} C_VEL
LIN {X 0,Y 447.91,Z 175.192,A -85,B 0,C 180,E1 -8855.082,E2 -8855.082} C_VEL
LIN {X 0,Y 447.724,Z 180.706,A -85,B 0,C 180,E1 -8856.13,E2 -8856.13} C_VEL
LIN {X 0,Y 451.01,Z 198.036,A -85,B 0,C 180,E1 -8856.598,E2 -8856.598} C_VEL
LIN {X 0,Y 450.098,Z 288.244,A -85,B 0,C 180,E1 -8858.115,E2 -8858.115} C_VEL
LIN {X 0,Y 449.768,Z 301.63,A -85,B 0,C 180,E1 -8858.525,E2 -8858.525} C_VEL
LIN {X 0,Y 449.296,Z 314.207,A -85,B 0,C 180,E1 -8859.092,E2 -8859.092} C_VEL
LIN {X 0,Y 448.805,Z 325.64,A -85,B 0,C 180,E1 -8859.792,E2 -8859.792} C_VEL
LIN {X 0,Y 448.207,Z 336.808,A -85,B 0,C 180,E1 -8860.668,E2 -8860.668} C_VEL
LIN {X 0,Y 447.606,Z 346.706,A -85,B 0,C 180,E1 -8861.631,E2 -8861.631} C_VEL
LIN {X 0,Y 447.071,Z 356.223,A -85,B 0,C 180,E1 -8862.768,E2 -8862.768} C_VEL
LIN {X 0,Y 446.512,Z 365.061,A -85,B 0,C 180,E1 -8864.082,E2 -8864.082} C_VEL
LIN {X 0,Y 446.081,Z 372.144,A -85,B 0,C 180,E1 -8865.38,E2 -8865.38} C_VEL
LIN {X 0,Y 445.774,Z 378.731,A -85,B 0,C 180,E1 -8866.893,E2 -8866.893} C_VEL
LIN {X 0,Y 445.568,Z 384.066,A -85,B 0,C 180,E1 -8868.513,E2 -8868.513} C_VEL
LIN {X 0,Y 445.428,Z 387.022,A -85,B 0,C 180,E1 -8869.694,E2 -8869.694} C_VEL
LIN {X 0,Y 445.307,Z 389.152,A -85,B 0,C 180,E1 -8870.856,E2 -8870.856} C_VEL
LIN {X 0,Y 445.201,Z 390.71,A -85,B 0,C 180,E1 -8872.12,E2 -8872.12} C_VEL
LIN {X 0,Y 445.147,Z 391.536,A -85,B 0,C 180,E1 -8873.628,E2 -8873.628} C_VEL
LIN {X 0,Y 445.21,Z 391.128,A -85,B 0,C 180,E1 -8875.371,E2 -8875.371} C_VEL
LIN {X 0,Y 445.228,Z 389.687,A -85,B 0,C 180,E1 -8876.783,E2 -8876.783} C_VEL
LIN {X 0,Y 445.425,Z 386.732,A -85,B 0,C 180,E1 -8878.431,E2 -8878.431} C_VEL
LIN {X 0,Y 445.538,Z 383.511,A -85,B 0,C 180,E1 -8879.685,E2 -8879.685} C_VEL
LIN {X 0,Y 445.786,Z 378.099,A -85,B 0,C 180,E1 -8881.261,E2 -8881.261} C_VEL
LIN {X 0,Y 446.14,Z 371.123,A -85,B 0,C 180,E1 -8882.819,E2 -8882.819} C_VEL
LIN {X 0,Y 446.51,Z 363.899,A -85,B 0,C 180,E1 -8884.103,E2 -8884.103} C_VEL
LIN {X 0,Y 446.995,Z 355.276,A -85,B 0,C 180,E1 -8885.343,E2 -8885.343} C_VEL
LIN {X 0,Y 447.477,Z 347.071,A -85,B 0,C 180,E1 -8886.319,E2 -8886.319} C_VEL
LIN {X 0,Y 447.019,Z 342.598,A -85,B 0,C 180,E1 -8886.802,E2 -8886.802} C_VEL
LIN {X 0,Y 443.53,Z 331.992,A -85,B 0,C 180,E1 -8887.869,E2 -8887.869} C_VEL
LIN {X 0,Y 441.995,Z 325.483,A -85,B 0,C 180,E1 -8888.414,E2 -8888.414} C_VEL
LIN {X 0,Y 441.863,Z 321.979,A -85,B 0,C 180,E1 -8888.657,E2 -8888.657} C_VEL
LIN {X 0,Y 442.421,Z 309.043,A -85,B 0,C 180,E1 -8889.382,E2 -8889.382} C_VEL
LIN {X 0,Y 442.846,Z 295.82,A -85,B 0,C 180,E1 -8889.9,E2 -8889.9} C_VEL
LIN {X 0,Y 443.122,Z 283.128,A -85,B 0,C 180,E1 -8890.215,E2 -8890.215} C_VEL
LIN {X 0,Y 443.903,Z 198.796,A -85,B 0,C 180,E1 -8891.631,E2 -8891.631} C_VEL
LIN {X 0,Y 440.654,Z 180.93,A -85,B 0,C 180,E1 -8892.092,E2 -8892.092} C_VEL
LIN {X 0,Y 440.728,Z 178.221,A -85,B 0,C 180,E1 -8892.591,E2 -8892.591} C_VEL
LIN {X 0,Y 441.368,Z 165.862,A -85,B 0,C 180,E1 -8895.241,E2 -8895.241} C_VEL
LIN {X 0,Y 439.492,Z 155.305,A -85,B 0,C 180,E1 -8897.724,E2 -8897.724} C_VEL
LIN {X 0,Y 439.496,Z 155.237,A -85,B 0,C 180,E1 -8900.799,E2 -8900.799} C_VEL
LIN {X 0,Y 439.615,Z 155.224,A -85,B 0,C 180,E1 -8903.576,E2 -8903.576} C_VEL
LIN {X 0,Y 439.637,Z 155.219,A -85,B 0,C 180,E1 -8907.252,E2 -8907.252} C_VEL
LIN {X 0,Y 439.759,Z 155.207,A -85,B 0,C 180,E1 -8910.001,E2 -8910.001} C_VEL
LIN {X 0,Y 439.638,Z 155.217,A -85,B 0,C 180,E1 -8912.75,E2 -8912.75} C_VEL
LIN {X 0,Y 439.603,Z 155.222,A -85,B 0,C 180,E1 -8916.426,E2 -8916.426} C_VEL
LIN {X 0,Y 439.495,Z 155.239,A -85,B 0,C 180,E1 -8919.203,E2 -8919.203} C_VEL
LIN {X 0,Y 439.464,Z 155.241,A -85,B 0,C 180,E1 -8922.938,E2 -8922.938} C_VEL
LIN {X 0,Y 439.445,Z 155.241,A -85,B 0,C 180,E1 -8926.349,E2 -8926.349} C_VEL
LIN {X 0,Y 439.401,Z 155.251,A -85,B 0,C 180,E1 -8929.627,E2 -8929.627} C_VEL
LIN {X 0,Y 439.363,Z 155.253,A -85,B 0,C 180,E1 -8932.576,E2 -8932.576} C_VEL
LIN {X 0,Y 439.397,Z 155.25,A -85,B 0,C 180,E1 -8935.586,E2 -8935.586} C_VEL
LIN {X 0,Y 439.416,Z 155.248,A -85,B 0,C 180,E1 -8938.674,E2 -8938.674} C_VEL
LIN {X 0,Y 439.367,Z 155.251,A -85,B 0,C 180,E1 -8942.031,E2 -8942.031} C_VEL
LIN {X 0,Y 439.391,Z 155.251,A -85,B 0,C 180,E1 -8945.34,E2 -8945.34} C_VEL
LIN {X 0,Y 439.376,Z 155.254,A -85,B 0,C 180,E1 -8948.596,E2 -8948.596} C_VEL
LIN {X 0,Y 439.388,Z 155.251,A -85,B 0,C 180,E1 -8951.257,E2 -8951.257} C_VEL
LIN {X 0,Y 439.398,Z 155.255,A -85,B 0,C 180,E1 -8954.73,E2 -8954.73} C_VEL
LIN {X 0,Y 439.383,Z 155.249,A -85,B 0,C 180,E1 -8957.795,E2 -8957.795} C_VEL
LIN {X 0,Y 439.357,Z 155.255,A -85,B 0,C 180,E1 -8960.22,E2 -8960.22} C_VEL
LIN {X 0,Y 439.371,Z 155.251,A -85,B 0,C 180,E1 -8963.713,E2 -8963.713} C_VEL
LIN {X 0,Y 439.371,Z 155.252,A -85,B 0,C 180,E1 -8967.054,E2 -8967.054} C_VEL
LIN {X 0,Y 439.376,Z 155.256,A -85,B 0,C 180,E1 -8970.274,E2 -8970.274} C_VEL
LIN {X 0,Y 439.381,Z 155.249,A -85,B 0,C 180,E1 -8973.394,E2 -8973.394} C_VEL
LIN {X 0,Y 439.383,Z 155.255,A -85,B 0,C 180,E1 -8976.43,E2 -8976.43} C_VEL
LIN {X 0,Y 439.387,Z 155.249,A -85,B 0,C 180,E1 -8979.398,E2 -8979.398} C_VEL
LIN {X 0,Y 439.423,Z 155.25,A -85,B 0,C 180,E1 -8982.31,E2 -8982.31} C_VEL
LIN {X 0,Y 439.444,Z 155.242,A -85,B 0,C 180,E1 -8985.174,E2 -8985.174} C_VEL
LIN {X 0,Y 439.483,Z 155.244,A -85,B 0,C 180,E1 -8988.002,E2 -8988.002} C_VEL
LIN {X 0,Y 439.502,Z 155.239,A -85,B 0,C 180,E1 -8991.726,E2 -8991.726} C_VEL
LIN {X 0,Y 439.597,Z 155.224,A -85,B 0,C 180,E1 -8994.496,E2 -8994.496} C_VEL
LIN {X 0,Y 439.626,Z 155.222,A -85,B 0,C 180,E1 -8998.168,E2 -8998.168} C_VEL
LIN {X 0,Y 439.668,Z 155.219,A -85,B 0,C 180,E1 -9000,E2 -9000} C_VEL
LIN {X 0,Y 439.615,Z 155.22,A -85,B 0,C 180,E1 -9002.749,E2 -9002.749} C_VEL
LIN {X 0,Y 439.551,Z 155.229,A -85,B 0,C 180,E1 -9006.427,E2 -9006.427} C_VEL
LIN {X 0,Y 439.479,Z 155.24,A -85,B 0,C 180,E1 -9009.202,E2 -9009.202} C_VEL
LIN {X 0,Y 439.466,Z 155.24,A -85,B 0,C 180,E1 -9012.938,E2 -9012.938} C_VEL
LIN {X 0,Y 439.445,Z 155.241,A -85,B 0,C 180,E1 -9016.347,E2 -9016.347} C_VEL
LIN {X 0,Y 439.401,Z 155.251,A -85,B 0,C 180,E1 -9019.627,E2 -9019.627} C_VEL
LIN {X 0,Y 439.363,Z 155.252,A -85,B 0,C 180,E1 -9022.576,E2 -9022.576} C_VEL
LIN {X 0,Y 439.355,Z 155.256,A -85,B 0,C 180,E1 -9025.588,E2 -9025.588} C_VEL
LIN {X 0,Y 439.378,Z 155.252,A -85,B 0,C 180,E1 -9028.677,E2 -9028.677} C_VEL
LIN {X 0,Y 439.344,Z 155.254,A -85,B 0,C 180,E1 -9032.024,E2 -9032.024} C_VEL
LIN {X 0,Y 439.386,Z 155.252,A -85,B 0,C 180,E1 -9035.338,E2 -9035.338} C_VEL
LIN {X 0,Y 439.351,Z 155.257,A -85,B 0,C 180,E1 -9038.599,E2 -9038.599} C_VEL
LIN {X 0,Y 439.346,Z 155.255,A -85,B 0,C 180,E1 -9042.211,E2 -9042.211} C_VEL
LIN {X 0,Y 439.377,Z 155.252,A -85,B 0,C 180,E1 -9045.267,E2 -9045.267} C_VEL
LIN {X 0,Y 439.35,Z 155.257,A -85,B 0,C 180,E1 -9049.015,E2 -9049.015} C_VEL
LIN {X 0,Y 439.328,Z 155.263,A -85,B 0,C 180,E1 -9052.562,E2 -9052.562} C_VEL
LIN {X 0,Y 439.328,Z 155.257,A -85,B 0,C 180,E1 -9055.951,E2 -9055.951} C_VEL
LIN {X 0,Y 439.343,Z 155.259,A -85,B 0,C 180,E1 -9059.21,E2 -9059.21} C_VEL
LIN {X 0,Y 439.333,Z 155.262,A -85,B 0,C 180,E1 -9062.36,E2 -9062.36} C_VEL
LIN {X 0,Y 439.42,Z 155.401,A -85,B 0,C 180,E1 -9064.177,E2 -9064.177} C_VEL
LIN {X 0,Y 441.739,Z 167.36,A -85,B 0,C 180,E1 -9066.785,E2 -9066.785} C_VEL
LIN {X 0,Y 441.531,Z 174.797,A -85,B 0,C 180,E1 -9068.279,E2 -9068.279} C_VEL
LIN {X 0,Y 440.529,Z 192.608,A -85,B 0,C 180,E1 -9071.79,E2 -9071.79} C_VEL
LIN {X 0,Y 440.541,Z 193.803,A -85,B 0,C 180,E1 -9071.944,E2 -9071.944} C_VEL
LIN {X 0,Y 443.937,Z 215.013,A -85,B 0,C 180,E1 -9072.468,E2 -9072.468} C_VEL
LIN {X 0,Y 443.034,Z 301.98,A -85,B 0,C 180,E1 -9073.941,E2 -9073.941} C_VEL
LIN {X 0,Y 442.575,Z 315.681,A -85,B 0,C 180,E1 -9074.367,E2 -9074.367} C_VEL
LIN {X 0,Y 442.006,Z 328.547,A -85,B 0,C 180,E1 -9074.966,E2 -9074.966} C_VEL
LIN {X 0,Y 441.452,Z 340.306,A -85,B 0,C 180,E1 -9075.713,E2 -9075.713} C_VEL
LIN {X 0,Y 440.799,Z 352.516,A -85,B 0,C 180,E1 -9076.711,E2 -9076.711} C_VEL
LIN {X 0,Y 440.229,Z 362.868,A -85,B 0,C 180,E1 -9077.787,E2 -9077.787} C_VEL
LIN {X 0,Y 439.61,Z 371.897,A -85,B 0,C 180,E1 -9078.939,E2 -9078.939} C_VEL
LIN {X 0,Y 439.137,Z 380.715,A -85,B 0,C 180,E1 -9080.325,E2 -9080.325} C_VEL
LIN {X 0,Y 438.77,Z 387.746,A -85,B 0,C 180,E1 -9081.711,E2 -9081.711} C_VEL
LIN {X 0,Y 438.515,Z 393.367,A -85,B 0,C 180,E1 -9083.095,E2 -9083.095} C_VEL
LIN {X 0,Y 438.404,Z 397.781,A -85,B 0,C 180,E1 -9084.48,E2 -9084.48} C_VEL
LIN {X 0,Y 438.345,Z 400.11,A -85,B 0,C 180,E1 -9085.401,E2 -9085.401} C_VEL
LIN {X 0,Y 438.26,Z 402.007,A -85,B 0,C 180,E1 -9086.321,E2 -9086.321} C_VEL
LIN {X 0,Y 438.294,Z 403.444,A -85,B 0,C 180,E1 -9087.242,E2 -9087.242} C_VEL
LIN {X 0,Y 438.274,Z 404.459,A -85,B 0,C 180,E1 -9088.161,E2 -9088.161} C_VEL
LIN {X 0,Y 438.229,Z 405.319,A -85,B 0,C 180,E1 -9089.999,E2 -9089.999} C_VEL
LIN {X 0,Y 438.231,Z 405.123,A -85,B 0,C 180,E1 -9090.918,E2 -9090.918} C_VEL
LIN {X 0,Y 438.274,Z 404.522,A -85,B 0,C 180,E1 -9091.837,E2 -9091.837} C_VEL
LIN {X 0,Y 438.294,Z 403.532,A -85,B 0,C 180,E1 -9092.756,E2 -9092.756} C_VEL
LIN {X 0,Y 438.259,Z 402.141,A -85,B 0,C 180,E1 -9093.677,E2 -9093.677} C_VEL
LIN {X 0,Y 438.419,Z 399.209,A -85,B 0,C 180,E1 -9095.057,E2 -9095.057} C_VEL
LIN {X 0,Y 438.466,Z 395.235,A -85,B 0,C 180,E1 -9096.441,E2 -9096.441} C_VEL
LIN {X 0,Y 438.735,Z 389.128,A -85,B 0,C 180,E1 -9098.056,E2 -9098.056} C_VEL
LIN {X 0,Y 439.086,Z 382.444,A -85,B 0,C 180,E1 -9099.442,E2 -9099.442} C_VEL
LIN {X 0,Y 439.532,Z 374.15,A -85,B 0,C 180,E1 -9100.828,E2 -9100.828} C_VEL
LIN {X 0,Y 440.183,Z 365.656,A -85,B 0,C 180,E1 -9101.978,E2 -9101.978} C_VEL
LIN {X 0,Y 440.848,Z 354.91,A -85,B 0,C 180,E1 -9103.154,E2 -9103.154} C_VEL
LIN {X 0,Y 441.435,Z 343.353,A -85,B 0,C 180,E1 -9104.168,E2 -9104.168} C_VEL
LIN {X 0,Y 442.052,Z 331.495,A -85,B 0,C 180,E1 -9104.971,E2 -9104.971} C_VEL
LIN {X 0,Y 442.697,Z 319.196,A -85,B 0,C 180,E1 -9105.597,E2 -9105.597} C_VEL
LIN {X 0,Y 443.103,Z 306.661,A -85,B 0,C 180,E1 -9106.055,E2 -9106.055} C_VEL
LIN {X 0,Y 443.434,Z 292.132,A -85,B 0,C 180,E1 -9106.367,E2 -9106.367} C_VEL
LIN {X 0,Y 444.151,Z 214.04,A -85,B 0,C 180,E1 -9107.688,E2 -9107.688} C_VEL
LIN {X 0,Y 440.658,Z 193.346,A -85,B 0,C 180,E1 -9108.231,E2 -9108.231} C_VEL
LIN {X 0,Y 440.714,Z 191.068,A -85,B 0,C 180,E1 -9108.597,E2 -9108.597} C_VEL
LIN {X 0,Y 441.8,Z 171.458,A -85,B 0,C 180,E1 -9112.443,E2 -9112.443} C_VEL
LIN {X 0,Y 441.614,Z 166.557,A -85,B 0,C 180,E1 -9113.443,E2 -9113.443} C_VEL
LIN {X 0,Y 439.461,Z 155.615,A -85,B 0,C 180,E1 -9115.82,E2 -9115.82} C_VEL
LIN {X 0,Y 439.415,Z 155.253,A -85,B 0,C 180,E1 -9116.063,E2 -9116.063} C_VEL
LIN {X 0,Y 439.373,Z 155.256,A -85,B 0,C 180,E1 -9118.675,E2 -9118.675} C_VEL
LIN {X 0,Y 439.348,Z 155.259,A -85,B 0,C 180,E1 -9122.025,E2 -9122.025} C_VEL
LIN {X 0,Y 439.381,Z 155.256,A -85,B 0,C 180,E1 -9125.337,E2 -9125.337} C_VEL
LIN {X 0,Y 439.347,Z 155.255,A -85,B 0,C 180,E1 -9128.597,E2 -9128.597} C_VEL
LIN {X 0,Y 439.356,Z 155.26,A -85,B 0,C 180,E1 -9131.251,E2 -9131.251} C_VEL
LIN {X 0,Y 439.367,Z 155.253,A -85,B 0,C 180,E1 -9134.731,E2 -9134.731} C_VEL
LIN {X 0,Y 439.338,Z 155.259,A -85,B 0,C 180,E1 -9137.788,E2 -9137.788} C_VEL
LIN {X 0,Y 439.348,Z 155.257,A -85,B 0,C 180,E1 -9141.401,E2 -9141.401} C_VEL
LIN {X 0,Y 439.384,Z 155.254,A -85,B 0,C 180,E1 -9144.842,E2 -9144.842} C_VEL
LIN {X 0,Y 439.342,Z 155.255,A -85,B 0,C 180,E1 -9148.137,E2 -9148.137} C_VEL
LIN {X 0,Y 439.369,Z 155.255,A -85,B 0,C 180,E1 -9151.323,E2 -9151.323} C_VEL
LIN {X 0,Y 439.353,Z 155.255,A -85,B 0,C 180,E1 -9154.411,E2 -9154.411} C_VEL
LIN {X 0,Y 439.35,Z 155.255,A -85,B 0,C 180,E1 -9157.423,E2 -9157.423} C_VEL
LIN {X 0,Y 439.429,Z 155.244,A -85,B 0,C 180,E1 -9160.662,E2 -9160.662} C_VEL
LIN {X 0,Y 439.447,Z 155.241,A -85,B 0,C 180,E1 -9164.224,E2 -9164.224} C_VEL
LIN {X 0,Y 439.469,Z 155.239,A -85,B 0,C 180,E1 -9168,E2 -9168} C_VEL
LIN {X 0,Y 439.49,Z 155.236,A -85,B 0,C 180,E1 -9171.725,E2 -9171.725} C_VEL
LIN {X 0,Y 439.593,Z 155.228,A -85,B 0,C 180,E1 -9174.495,E2 -9174.495} C_VEL
LIN {X 0,Y 439.616,Z 155.223,A -85,B 0,C 180,E1 -9178.167,E2 -9178.167} C_VEL
LIN {X 0,Y 439.582,Z 155.229,A -85,B 0,C 180,E1 -9180.916,E2 -9180.916} C_VEL
LIN {X 0,Y 439.595,Z 155.225,A -85,B 0,C 180,E1 -9182.749,E2 -9182.749} C_VEL
LIN {X 0,Y 439.581,Z 155.229,A -85,B 0,C 180,E1 -9186.425,E2 -9186.425} C_VEL
LIN {X 0,Y 439.468,Z 155.239,A -85,B 0,C 180,E1 -9189.202,E2 -9189.202} C_VEL
LIN {X 0,Y 439.451,Z 155.244,A -85,B 0,C 180,E1 -9192.938,E2 -9192.938} C_VEL
LIN {X 0,Y 439.431,Z 155.25,A -85,B 0,C 180,E1 -9196.348,E2 -9196.348} C_VEL
LIN {X 0,Y 439.388,Z 155.252,A -85,B 0,C 180,E1 -9199.626,E2 -9199.626} C_VEL
LIN {X 0,Y 439.349,Z 155.26,A -85,B 0,C 180,E1 -9202.576,E2 -9202.576} C_VEL
LIN {X 0,Y 439.351,Z 155.256,A -85,B 0,C 180,E1 -9205.588,E2 -9205.588} C_VEL
LIN {X 0,Y 439.369,Z 155.257,A -85,B 0,C 180,E1 -9208.676,E2 -9208.676} C_VEL
LIN {X 0,Y 439.435,Z 155.463,A -85,B 0,C 180,E1 -9210.479,E2 -9210.479} C_VEL
LIN {X 0,Y 441.361,Z 165.716,A -85,B 0,C 180,E1 -9212.778,E2 -9212.778} C_VEL
LIN {X 0,Y 440.831,Z 179.701,A -85,B 0,C 180,E1 -9215.658,E2 -9215.658} C_VEL
LIN {X 0,Y 440.851,Z 181.08,A -85,B 0,C 180,E1 -9215.842,E2 -9215.842} C_VEL
LIN {X 0,Y 444.383,Z 199.623,A -85,B 0,C 180,E1 -9216.339,E2 -9216.339} C_VEL
LIN {X 0,Y 443.293,Z 288.802,A -85,B 0,C 180,E1 -9217.866,E2 -9217.866} C_VEL
LIN {X 0,Y 442.945,Z 302.253,A -85,B 0,C 180,E1 -9218.29,E2 -9218.29} C_VEL
LIN {X 0,Y 442.422,Z 315.107,A -85,B 0,C 180,E1 -9218.89,E2 -9218.89} C_VEL
LIN {X 0,Y 441.903,Z 326.563,A -85,B 0,C 180,E1 -9219.618,E2 -9219.618} C_VEL
LIN {X 0,Y 441.239,Z 337.77,A -85,B 0,C 180,E1 -9220.522,E2 -9220.522} C_VEL
LIN {X 0,Y 440.655,Z 347.029,A -85,B 0,C 180,E1 -9221.447,E2 -9221.447} C_VEL
LIN {X 0,Y 440.109,Z 356.225,A -85,B 0,C 180,E1 -9222.565,E2 -9222.565} C_VEL
LIN {X 0,Y 439.606,Z 363.904,A -85,B 0,C 180,E1 -9223.699,E2 -9223.699} C_VEL
LIN {X 0,Y 439.118,Z 371.094,A -85,B 0,C 180,E1 -9224.991,E2 -9224.991} C_VEL
LIN {X 0,Y 438.778,Z 377.681,A -85,B 0,C 180,E1 -9226.472,E2 -9226.472} C_VEL
LIN {X 0,Y 438.603,Z 382.066,A -85,B 0,C 180,E1 -9227.704,E2 -9227.704} C_VEL
LIN {X 0,Y 438.458,Z 385.524,A -85,B 0,C 180,E1 -9228.917,E2 -9228.917} C_VEL
LIN {X 0,Y 438.245,Z 388.53,A -85,B 0,C 180,E1 -9230.332,E2 -9230.332} C_VEL
LIN {X 0,Y 438.133,Z 390.588,A -85,B 0,C 180,E1 -9231.812,E2 -9231.812} C_VEL
LIN {X 0,Y 438.071,Z 391.644,A -85,B 0,C 180,E1 -9233.589,E2 -9233.589} C_VEL
LIN {X 0,Y 438.09,Z 391.493,A -85,B 0,C 180,E1 -9234.9,E2 -9234.9} C_VEL
LIN {X 0,Y 438.113,Z 390.151,A -85,B 0,C 180,E1 -9236.527,E2 -9236.527} C_VEL
LIN {X 0,Y 438.299,Z 387.457,A -85,B 0,C 180,E1 -9238.193,E2 -9238.193} C_VEL
LIN {X 0,Y 438.435,Z 384.13,A -85,B 0,C 180,E1 -9239.575,E2 -9239.575} C_VEL
LIN {X 0,Y 438.711,Z 378.542,A -85,B 0,C 180,E1 -9241.278,E2 -9241.278} C_VEL
LIN {X 0,Y 439.068,Z 371.642,A -85,B 0,C 180,E1 -9242.86,E2 -9242.86} C_VEL
LIN {X 0,Y 439.457,Z 364.425,A -85,B 0,C 180,E1 -9244.179,E2 -9244.179} C_VEL
LIN {X 0,Y 439.999,Z 355.728,A -85,B 0,C 180,E1 -9245.464,E2 -9245.464} C_VEL
LIN {X 0,Y 440.582,Z 346.022,A -85,B 0,C 180,E1 -9246.623,E2 -9246.623} C_VEL
LIN {X 0,Y 441.159,Z 335.72,A -85,B 0,C 180,E1 -9247.622,E2 -9247.622} C_VEL
LIN {X 0,Y 441.779,Z 323.794,A -85,B 0,C 180,E1 -9248.539,E2 -9248.539} C_VEL
LIN {X 0,Y 441.863,Z 321.979,A -85,B 0,C 180,E1 -9248.657,E2 -9248.657} C_VEL
LIN {X 0,Y 441.501,Z 316.714,A -85,B 0,C 180,E1 -9249,E2 -9249} C_VEL
LIN {X 0,Y 439.167,Z 308.035,A -85,B 0,C 180,E1 -9249.54,E2 -9249.54} C_VEL
LIN {X 0,Y 436.693,Z 299.121,A -85,B 0,C 180,E1 -9250.004,E2 -9250.004} C_VEL
LIN {X 0,Y 436.046,Z 293.487,A -85,B 0,C 180,E1 -9250.217,E2 -9250.217} C_VEL
LIN {X 0,Y 436.317,Z 280.608,A -85,B 0,C 180,E1 -9250.506,E2 -9250.506} C_VEL
LIN {X 0,Y 437.12,Z 199.697,A -85,B 0,C 180,E1 -9251.884,E2 -9251.884} C_VEL
LIN {X 0,Y 433.737,Z 180.943,A -85,B 0,C 180,E1 -9252.375,E2 -9252.375} C_VEL
LIN {X 0,Y 433.952,Z 175.301,A -85,B 0,C 180,E1 -9253.537,E2 -9253.537} C_VEL
LIN {X 0,Y 434.352,Z 166.427,A -85,B 0,C 180,E1 -9255.477,E2 -9255.477} C_VEL
LIN {X 0,Y 432.462,Z 156.195,A -85,B 0,C 180,E1 -9257.924,E2 -9257.924} C_VEL
LIN {X 0,Y 432.488,Z 156.112,A -85,B 0,C 180,E1 -9261.591,E2 -9261.591} C_VEL
LIN {X 0,Y 432.594,Z 156.097,A -85,B 0,C 180,E1 -9264.407,E2 -9264.407} C_VEL
LIN {X 0,Y 432.6,Z 156.097,A -85,B 0,C 180,E1 -9268.139,E2 -9268.139} C_VEL
LIN {X 0,Y 432.729,Z 156.083,A -85,B 0,C 180,E1 -9270.001,E2 -9270.001} C_VEL
LIN {X 0,Y 432.59,Z 156.096,A -85,B 0,C 180,E1 -9272.795,E2 -9272.795} C_VEL
LIN {X 0,Y 432.553,Z 156.1,A -85,B 0,C 180,E1 -9276.531,E2 -9276.531} C_VEL
LIN {X 0,Y 432.438,Z 156.12,A -85,B 0,C 180,E1 -9279.354,E2 -9279.354} C_VEL
LIN {X 0,Y 432.429,Z 156.116,A -85,B 0,C 180,E1 -9282.804,E2 -9282.804} C_VEL
LIN {X 0,Y 432.411,Z 156.118,A -85,B 0,C 180,E1 -9286.479,E2 -9286.479} C_VEL
LIN {X 0,Y 432.337,Z 156.128,A -85,B 0,C 180,E1 -9289.961,E2 -9289.961} C_VEL
LIN {X 0,Y 432.317,Z 156.134,A -85,B 0,C 180,E1 -9292.965,E2 -9292.965} C_VEL
LIN {X 0,Y 432.36,Z 156.124,A -85,B 0,C 180,E1 -9296.033,E2 -9296.033} C_VEL
LIN {X 0,Y 432.342,Z 156.133,A -85,B 0,C 180,E1 -9299.188,E2 -9299.188} C_VEL
LIN {X 0,Y 432.321,Z 156.13,A -85,B 0,C 180,E1 -9302.444,E2 -9302.444} C_VEL
LIN {X 0,Y 432.342,Z 156.127,A -85,B 0,C 180,E1 -9305.632,E2 -9305.632} C_VEL
LIN {X 0,Y 432.338,Z 156.132,A -85,B 0,C 180,E1 -9308.715,E2 -9308.715} C_VEL
LIN {X 0,Y 432.332,Z 156.128,A -85,B 0,C 180,E1 -9311.798,E2 -9311.798} C_VEL
LIN {X 0,Y 432.333,Z 156.13,A -85,B 0,C 180,E1 -9314.348,E2 -9314.348} C_VEL
LIN {X 0,Y 432.315,Z 156.134,A -85,B 0,C 180,E1 -9317.017,E2 -9317.017} C_VEL
LIN {X 0,Y 432.312,Z 156.13,A -85,B 0,C 180,E1 -9319.825,E2 -9319.825} C_VEL
LIN {X 0,Y 432.304,Z 156.134,A -85,B 0,C 180,E1 -9323.022,E2 -9323.022} C_VEL
LIN {X 0,Y 432.359,Z 156.126,A -85,B 0,C 180,E1 -9325.997,E2 -9325.997} C_VEL
LIN {X 0,Y 432.346,Z 156.126,A -85,B 0,C 180,E1 -9329.491,E2 -9329.491} C_VEL
LIN {X 0,Y 432.343,Z 156.128,A -85,B 0,C 180,E1 -9331.874,E2 -9331.874} C_VEL
LIN {X 0,Y 432.377,Z 156.122,A -85,B 0,C 180,E1 -9335.539,E2 -9335.539} C_VEL
LIN {X 0,Y 432.349,Z 156.126,A -85,B 0,C 180,E1 -9339.046,E2 -9339.046} C_VEL
LIN {X 0,Y 432.371,Z 156.128,A -85,B 0,C 180,E1 -9342.011,E2 -9342.011} C_VEL
LIN {X 0,Y 432.392,Z 156.12,A -85,B 0,C 180,E1 -9344.927,E2 -9344.927} C_VEL
LIN {X 0,Y 432.459,Z 156.116,A -85,B 0,C 180,E1 -9347.804,E2 -9347.804} C_VEL
LIN {X 0,Y 432.462,Z 156.114,A -85,B 0,C 180,E1 -9351.59,E2 -9351.59} C_VEL
LIN {X 0,Y 432.571,Z 156.1,A -85,B 0,C 180,E1 -9354.406,E2 -9354.406} C_VEL
LIN {X 0,Y 432.595,Z 156.099,A -85,B 0,C 180,E1 -9358.138,E2 -9358.138} C_VEL
LIN {X 0,Y 432.62,Z 156.097,A -85,B 0,C 180,E1 -9360,E2 -9360} C_VEL
LIN {X 0,Y 432.569,Z 156.098,A -85,B 0,C 180,E1 -9362.794,E2 -9362.794} C_VEL
LIN {X 0,Y 432.507,Z 156.106,A -85,B 0,C 180,E1 -9366.532,E2 -9366.532} C_VEL
LIN {X 0,Y 432.425,Z 156.121,A -85,B 0,C 180,E1 -9369.354,E2 -9369.354} C_VEL
LIN {X 0,Y 432.432,Z 156.116,A -85,B 0,C 180,E1 -9372.803,E2 -9372.803} C_VEL
LIN {X 0,Y 432.396,Z 156.12,A -85,B 0,C 180,E1 -9376.47,E2 -9376.47} C_VEL
LIN {X 0,Y 432.336,Z 156.128,A -85,B 0,C 180,E1 -9379.961,E2 -9379.961} C_VEL
LIN {X 0,Y 432.311,Z 156.134,A -85,B 0,C 180,E1 -9382.965,E2 -9382.965} C_VEL
LIN {X 0,Y 432.307,Z 156.131,A -85,B 0,C 180,E1 -9386.037,E2 -9386.037} C_VEL
LIN {X 0,Y 432.316,Z 156.137,A -85,B 0,C 180,E1 -9389.19,E2 -9389.19} C_VEL
LIN {X 0,Y 432.306,Z 156.132,A -85,B 0,C 180,E1 -9392.445,E2 -9392.445} C_VEL
LIN {X 0,Y 432.334,Z 156.128,A -85,B 0,C 180,E1 -9395.819,E2 -9395.819} C_VEL
LIN {X 0,Y 432.315,Z 156.134,A -85,B 0,C 180,E1 -9398.71,E2 -9398.71} C_VEL
LIN {X 0,Y 432.302,Z 156.131,A -85,B 0,C 180,E1 -9401.801,E2 -9401.801} C_VEL
LIN {X 0,Y 432.336,Z 156.129,A -85,B 0,C 180,E1 -9404.347,E2 -9404.347} C_VEL
LIN {X 0,Y 432.303,Z 156.136,A -85,B 0,C 180,E1 -9407.019,E2 -9407.019} C_VEL
LIN {X 0,Y 432.29,Z 156.133,A -85,B 0,C 180,E1 -9409.828,E2 -9409.828} C_VEL
LIN {X 0,Y 432.287,Z 156.136,A -85,B 0,C 180,E1 -9413.02,E2 -9413.02} C_VEL
LIN {X 0,Y 432.308,Z 156.132,A -85,B 0,C 180,E1 -9416.007,E2 -9416.007} C_VEL
LIN {X 0,Y 432.334,Z 156.131,A -85,B 0,C 180,E1 -9419.494,E2 -9419.494} C_VEL
LIN {X 0,Y 432.315,Z 156.136,A -85,B 0,C 180,E1 -9421.871,E2 -9421.871} C_VEL
LIN {X 0,Y 432.383,Z 156.322,A -85,B 0,C 180,E1 -9423.968,E2 -9423.968} C_VEL
LIN {X 0,Y 434.749,Z 168.513,A -85,B 0,C 180,E1 -9426.668,E2 -9426.668} C_VEL
LIN {X 0,Y 434.653,Z 174.609,A -85,B 0,C 180,E1 -9427.917,E2 -9427.917} C_VEL
LIN {X 0,Y 433.584,Z 192.817,A -85,B 0,C 180,E1 -9431.555,E2 -9431.555} C_VEL
LIN {X 0,Y 433.614,Z 194.079,A -85,B 0,C 180,E1 -9431.679,E2 -9431.679} C_VEL
LIN {X 0,Y 437.146,Z 215.649,A -85,B 0,C 180,E1 -9432.213,E2 -9432.213} C_VEL
LIN {X 0,Y 436.21,Z 301.233,A -85,B 0,C 180,E1 -9433.683,E2 -9433.683} C_VEL
LIN {X 0,Y 435.768,Z 314.379,A -85,B 0,C 180,E1 -9434.086,E2 -9434.086} C_VEL
LIN {X 0,Y 435.223,Z 327.073,A -85,B 0,C 180,E1 -9434.667,E2 -9434.667} C_VEL
LIN {X 0,Y 434.636,Z 338.38,A -85,B 0,C 180,E1 -9435.365,E2 -9435.365} C_VEL
LIN {X 0,Y 434.002,Z 349.66,A -85,B 0,C 180,E1 -9436.263,E2 -9436.263} C_VEL
LIN {X 0,Y 433.411,Z 360.576,A -85,B 0,C 180,E1 -9437.354,E2 -9437.354} C_VEL
LIN {X 0,Y 432.769,Z 370.035,A -85,B 0,C 180,E1 -9438.524,E2 -9438.524} C_VEL
LIN {X 0,Y 432.189,Z 379.15,A -85,B 0,C 180,E1 -9439.932,E2 -9439.932} C_VEL
LIN {X 0,Y 431.745,Z 386.492,A -85,B 0,C 180,E1 -9441.339,E2 -9441.339} C_VEL
LIN {X 0,Y 431.541,Z 391.46,A -85,B 0,C 180,E1 -9442.513,E2 -9442.513} C_VEL
LIN {X 0,Y 431.302,Z 396.526,A -85,B 0,C 180,E1 -9444,E2 -9444} C_VEL
LIN {X 0,Y 431.276,Z 399.968,A -85,B 0,C 180,E1 -9445.325,E2 -9445.325} C_VEL
LIN {X 0,Y 431.169,Z 401.871,A -85,B 0,C 180,E1 -9446.261,E2 -9446.261} C_VEL
LIN {X 0,Y 431.19,Z 403.317,A -85,B 0,C 180,E1 -9447.196,E2 -9447.196} C_VEL
LIN {X 0,Y 431.197,Z 404.338,A -85,B 0,C 180,E1 -9448.131,E2 -9448.131} C_VEL
LIN {X 0,Y 431.144,Z 405.207,A -85,B 0,C 180,E1 -9449.999,E2 -9449.999} C_VEL
LIN {X 0,Y 431.149,Z 405.018,A -85,B 0,C 180,E1 -9450.933,E2 -9450.933} C_VEL
LIN {X 0,Y 431.197,Z 404.422,A -85,B 0,C 180,E1 -9451.867,E2 -9451.867} C_VEL
LIN {X 0,Y 431.19,Z 403.433,A -85,B 0,C 180,E1 -9452.802,E2 -9452.802} C_VEL
LIN {X 0,Y 431.168,Z 402.047,A -85,B 0,C 180,E1 -9453.737,E2 -9453.737} C_VEL
LIN {X 0,Y 431.331,Z 399.119,A -85,B 0,C 180,E1 -9455.14,E2 -9455.14} C_VEL
LIN {X 0,Y 431.386,Z 395.152,A -85,B 0,C 180,E1 -9456.547,E2 -9456.547} C_VEL
LIN {X 0,Y 431.689,Z 389.054,A -85,B 0,C 180,E1 -9458.189,E2 -9458.189} C_VEL
LIN {X 0,Y 432.066,Z 382.376,A -85,B 0,C 180,E1 -9459.596,E2 -9459.596} C_VEL
LIN {X 0,Y 432.547,Z 374.088,A -85,B 0,C 180,E1 -9461.005,E2 -9461.005} C_VEL
LIN {X 0,Y 433.224,Z 365.615,A -85,B 0,C 180,E1 -9462.174,E2 -9462.174} C_VEL
LIN {X 0,Y 433.866,Z 355.711,A -85,B 0,C 180,E1 -9463.288,E2 -9463.288} C_VEL
LIN {X 0,Y 434.457,Z 344.808,A -85,B 0,C 180,E1 -9464.281,E2 -9464.281} C_VEL
LIN {X 0,Y 435.082,Z 333.494,A -85,B 0,C 180,E1 -9465.097,E2 -9465.097} C_VEL
LIN {X 0,Y 435.763,Z 321.961,A -85,B 0,C 180,E1 -9465.732,E2 -9465.732} C_VEL
LIN {X 0,Y 436.233,Z 308.773,A -85,B 0,C 180,E1 -9466.254,E2 -9466.254} C_VEL
LIN {X 0,Y 436.61,Z 296.108,A -85,B 0,C 180,E1 -9466.57,E2 -9466.57} C_VEL
LIN {X 0,Y 437.452,Z 215.124,A -85,B 0,C 180,E1 -9467.964,E2 -9467.964} C_VEL
LIN {X 0,Y 433.77,Z 193.424,A -85,B 0,C 180,E1 -9468.539,E2 -9468.539} C_VEL
LIN {X 0,Y 433.754,Z 192.245,A -85,B 0,C 180,E1 -9468.678,E2 -9468.678} C_VEL
LIN {X 0,Y 434.889,Z 172.683,A -85,B 0,C 180,E1 -9472.569,E2 -9472.569} C_VEL
LIN {X 0,Y 434.665,Z 167.778,A -85,B 0,C 180,E1 -9473.588,E2 -9473.588} C_VEL
LIN {X 0,Y 432.429,Z 156.4,A -85,B 0,C 180,E1 -9476.118,E2 -9476.118} C_VEL
LIN {X 0,Y 432.316,Z 156.135,A -85,B 0,C 180,E1 -9476.604,E2 -9476.604} C_VEL
LIN {X 0,Y 432.311,Z 156.135,A -85,B 0,C 180,E1 -9479.188,E2 -9479.188} C_VEL
LIN {X 0,Y 432.311,Z 156.133,A -85,B 0,C 180,E1 -9482.442,E2 -9482.442} C_VEL
LIN {X 0,Y 432.327,Z 156.134,A -85,B 0,C 180,E1 -9485.817,E2 -9485.817} C_VEL
LIN {X 0,Y 432.293,Z 156.14,A -85,B 0,C 180,E1 -9489.347,E2 -9489.347} C_VEL
LIN {X 0,Y 432.295,Z 156.136,A -85,B 0,C 180,E1 -9491.799,E2 -9491.799} C_VEL
LIN {X 0,Y 432.324,Z 156.129,A -85,B 0,C 180,E1 -9494.346,E2 -9494.346} C_VEL
LIN {X 0,Y 432.292,Z 156.137,A -85,B 0,C 180,E1 -9497.017,E2 -9497.017} C_VEL
LIN {X 0,Y 432.279,Z 156.137,A -85,B 0,C 180,E1 -9499.827,E2 -9499.827} C_VEL
LIN {X 0,Y 432.289,Z 156.135,A -85,B 0,C 180,E1 -9503.02,E2 -9503.02} C_VEL
LIN {X 0,Y 432.323,Z 156.128,A -85,B 0,C 180,E1 -9506.001,E2 -9506.001} C_VEL
LIN {X 0,Y 432.327,Z 156.131,A -85,B 0,C 180,E1 -9509.491,E2 -9509.491} C_VEL
LIN {X 0,Y 432.308,Z 156.13,A -85,B 0,C 180,E1 -9511.871,E2 -9511.871} C_VEL
LIN {X 0,Y 432.31,Z 156.137,A -85,B 0,C 180,E1 -9514.996,E2 -9514.996} C_VEL
LIN {X 0,Y 432.345,Z 156.126,A -85,B 0,C 180,E1 -9518.045,E2 -9518.045} C_VEL
LIN {X 0,Y 432.371,Z 156.123,A -85,B 0,C 180,E1 -9521.029,E2 -9521.029} C_VEL
LIN {X 0,Y 432.416,Z 156.116,A -85,B 0,C 180,E1 -9523.96,E2 -9523.96} C_VEL
LIN {X 0,Y 432.445,Z 156.113,A -85,B 0,C 180,E1 -9527.803,E2 -9527.803} C_VEL
LIN {X 0,Y 432.45,Z 156.113,A -85,B 0,C 180,E1 -9531.589,E2 -9531.589} C_VEL
LIN {X 0,Y 432.57,Z 156.102,A -85,B 0,C 180,E1 -9534.405,E2 -9534.405} C_VEL
LIN {X 0,Y 432.585,Z 156.099,A -85,B 0,C 180,E1 -9538.138,E2 -9538.138} C_VEL
LIN {X 0,Y 432.542,Z 156.106,A -85,B 0,C 180,E1 -9540.931,E2 -9540.931} C_VEL
LIN {X 0,Y 432.548,Z 156.102,A -85,B 0,C 180,E1 -9542.793,E2 -9542.793} C_VEL
LIN {X 0,Y 432.569,Z 156.099,A -85,B 0,C 180,E1 -9545.594,E2 -9545.594} C_VEL
LIN {X 0,Y 432.446,Z 156.119,A -85,B 0,C 180,E1 -9548.41,E2 -9548.41} C_VEL
LIN {X 0,Y 432.439,Z 156.119,A -85,B 0,C 180,E1 -9552.197,E2 -9552.197} C_VEL
LIN {X 0,Y 432.415,Z 156.122,A -85,B 0,C 180,E1 -9556.039,E2 -9556.039} C_VEL
LIN {X 0,Y 432.373,Z 156.125,A -85,B 0,C 180,E1 -9559.485,E2 -9559.485} C_VEL
LIN {X 0,Y 432.298,Z 156.136,A -85,B 0,C 180,E1 -9562.965,E2 -9562.965} C_VEL
LIN {X 0,Y 432.303,Z 156.138,A -85,B 0,C 180,E1 -9566.036,E2 -9566.036} C_VEL
LIN {X 0,Y 432.312,Z 156.137,A -85,B 0,C 180,E1 -9569.189,E2 -9569.189} C_VEL
LIN {X 0,Y 432.384,Z 156.268,A -85,B 0,C 180,E1 -9570.189,E2 -9570.189} C_VEL
LIN {X 0,Y 434.397,Z 166.724,A -85,B 0,C 180,E1 -9572.59,E2 -9572.59} C_VEL
LIN {X 0,Y 434.002,Z 178.627,A -85,B 0,C 180,E1 -9575.09,E2 -9575.09} C_VEL
LIN {X 0,Y 433.927,Z 180.755,A -85,B 0,C 180,E1 -9575.488,E2 -9575.488} C_VEL
LIN {X 0,Y 435.377,Z 188.272,A -85,B 0,C 180,E1 -9575.73,E2 -9575.73} C_VEL
LIN {X 0,Y 437.615,Z 200.299,A -85,B 0,C 180,E1 -9576.049,E2 -9576.049} C_VEL
LIN {X 0,Y 436.523,Z 288.845,A -85,B 0,C 180,E1 -9577.592,E2 -9577.592} C_VEL
LIN {X 0,Y 436.143,Z 302.521,A -85,B 0,C 180,E1 -9578.03,E2 -9578.03} C_VEL
LIN {X 0,Y 435.603,Z 315.353,A -85,B 0,C 180,E1 -9578.642,E2 -9578.642} C_VEL
LIN {X 0,Y 435.01,Z 327.264,A -85,B 0,C 180,E1 -9579.415,E2 -9579.415} C_VEL
LIN {X 0,Y 434.31,Z 338.388,A -85,B 0,C 180,E1 -9580.336,E2 -9580.336} C_VEL
LIN {X 0,Y 433.627,Z 348.828,A -85,B 0,C 180,E1 -9581.42,E2 -9581.42} C_VEL
LIN {X 0,Y 432.956,Z 358.924,A -85,B 0,C 180,E1 -9582.736,E2 -9582.736} C_VEL
LIN {X 0,Y 432.4,Z 366.873,A -85,B 0,C 180,E1 -9584.013,E2 -9584.013} C_VEL
LIN {X 0,Y 431.967,Z 373.372,A -85,B 0,C 180,E1 -9585.288,E2 -9585.288} C_VEL
LIN {X 0,Y 431.637,Z 379.735,A -85,B 0,C 180,E1 -9586.857,E2 -9586.857} C_VEL
LIN {X 0,Y 431.391,Z 384.894,A -85,B 0,C 180,E1 -9588.538,E2 -9588.538} C_VEL
LIN {X 0,Y 431.19,Z 388.152,A -85,B 0,C 180,E1 -9590,E2 -9590} C_VEL
LIN {X 0,Y 431.059,Z 390.653,A -85,B 0,C 180,E1 -9591.718,E2 -9591.718} C_VEL
LIN {X 0,Y 430.97,Z 391.6,A -85,B 0,C 180,E1 -9593.04,E2 -9593.04} C_VEL
LIN {X 0,Y 431,Z 391.71,A -85,B 0,C 180,E1 -9594.618,E2 -9594.618} C_VEL
LIN {X 0,Y 431.021,Z 390.529,A -85,B 0,C 180,E1 -9596.333,E2 -9596.333} C_VEL
LIN {X 0,Y 431.159,Z 388.135,A -85,B 0,C 180,E1 -9597.952,E2 -9597.952} C_VEL
LIN {X 0,Y 431.36,Z 384.201,A -85,B 0,C 180,E1 -9599.665,E2 -9599.665} C_VEL
LIN {X 0,Y 431.627,Z 379.369,A -85,B 0,C 180,E1 -9601.189,E2 -9601.189} C_VEL
LIN {X 0,Y 431.933,Z 373.435,A -85,B 0,C 180,E1 -9602.637,E2 -9602.637} C_VEL
LIN {X 0,Y 432.302,Z 366.642,A -85,B 0,C 180,E1 -9603.965,E2 -9603.965} C_VEL
LIN {X 0,Y 432.857,Z 357.54,A -85,B 0,C 180,E1 -9605.398,E2 -9605.398} C_VEL
LIN {X 0,Y 433.498,Z 348.081,A -85,B 0,C 180,E1 -9606.598,E2 -9606.598} C_VEL
LIN {X 0,Y 434.161,Z 337.294,A -85,B 0,C 180,E1 -9607.693,E2 -9607.693} C_VEL
LIN {X 0,Y 434.756,Z 326.815,A -85,B 0,C 180,E1 -9608.548,E2 -9608.548} C_VEL
LIN {X 0,Y 435.352,Z 314.108,A -85,B 0,C 180,E1 -9609.358,E2 -9609.358} C_VEL
LIN {X 0,Y 435.817,Z 300.663,A -85,B 0,C 180,E1 -9609.974,E2 -9609.974} C_VEL
LIN {X 0,Y 436.046,Z 293.487,A -85,B 0,C 180,E1 -9610.217,E2 -9610.217} C_VEL
LIN {X 0,Y 435.433,Z 287.774,A -85,B 0,C 180,E1 -9610.405,E2 -9610.405} C_VEL
LIN {X 0,Y 430.217,Z 269.073,A -85,B 0,C 180,E1 -9610.939,E2 -9610.939} C_VEL
LIN {X 0,Y 429.696,Z 263.255,A -85,B 0,C 180,E1 -9611.055,E2 -9611.055} C_VEL
LIN {X 0,Y 430.338,Z 200.643,A -85,B 0,C 180,E1 -9612.14,E2 -9612.14} C_VEL
LIN {X 0,Y 426.813,Z 181.334,A -85,B 0,C 180,E1 -9612.649,E2 -9612.649} C_VEL
LIN {X 0,Y 426.758,Z 180.326,A -85,B 0,C 180,E1 -9612.776,E2 -9612.776} C_VEL
LIN {X 0,Y 427.427,Z 168.032,A -85,B 0,C 180,E1 -9615.479,E2 -9615.479} C_VEL
LIN {X 0,Y 425.408,Z 157.066,A -85,B 0,C 180,E1 -9618.144,E2 -9618.144} C_VEL
LIN {X 0,Y 425.536,Z 156.977,A -85,B 0,C 180,E1 -9622.277,E2 -9622.277} C_VEL
LIN {X 0,Y 425.551,Z 156.975,A -85,B 0,C 180,E1 -9624.314,E2 -9624.314} C_VEL
LIN {X 0,Y 425.57,Z 156.974,A -85,B 0,C 180,E1 -9628.108,E2 -9628.108} C_VEL
LIN {X 0,Y 425.699,Z 156.958,A -85,B 0,C 180,E1 -9630.001,E2 -9630.001} C_VEL
LIN {X 0,Y 425.543,Z 156.973,A -85,B 0,C 180,E1 -9632.841,E2 -9632.841} C_VEL
LIN {X 0,Y 425.545,Z 156.98,A -85,B 0,C 180,E1 -9635.688,E2 -9635.688} C_VEL
LIN {X 0,Y 425.406,Z 156.99,A -85,B 0,C 180,E1 -9638.552,E2 -9638.552} C_VEL
LIN {X 0,Y 425.411,Z 156.99,A -85,B 0,C 180,E1 -9642.403,E2 -9642.403} C_VEL
LIN {X 0,Y 425.387,Z 156.993,A -85,B 0,C 180,E1 -9646.313,E2 -9646.313} C_VEL
LIN {X 0,Y 425.327,Z 157.004,A -85,B 0,C 180,E1 -9649.636,E2 -9649.636} C_VEL
LIN {X 0,Y 425.304,Z 157.009,A -85,B 0,C 180,E1 -9653.366,E2 -9653.366} C_VEL
LIN {X 0,Y 425.346,Z 157.001,A -85,B 0,C 180,E1 -9656.845,E2 -9656.845} C_VEL
LIN {X 0,Y 425.29,Z 157.006,A -85,B 0,C 180,E1 -9659.72,E2 -9659.72} C_VEL
LIN {X 0,Y 425.281,Z 157.013,A -85,B 0,C 180,E1 -9663.049,E2 -9663.049} C_VEL
LIN {X 0,Y 425.28,Z 157.006,A -85,B 0,C 180,E1 -9665.929,E2 -9665.929} C_VEL
LIN {X 0,Y 425.282,Z 157.012,A -85,B 0,C 180,E1 -9669.041,E2 -9669.041} C_VEL
LIN {X 0,Y 425.289,Z 157.005,A -85,B 0,C 180,E1 -9671.959,E2 -9671.959} C_VEL
LIN {X 0,Y 425.284,Z 157.007,A -85,B 0,C 180,E1 -9675.284,E2 -9675.284} C_VEL
LIN {X 0,Y 425.264,Z 157.015,A -85,B 0,C 180,E1 -9678.621,E2 -9678.621} C_VEL
LIN {X 0,Y 425.28,Z 157.008,A -85,B 0,C 180,E1 -9681.1,E2 -9681.1} C_VEL
LIN {X 0,Y 425.298,Z 157.01,A -85,B 0,C 180,E1 -9684.665,E2 -9684.665} C_VEL
LIN {X 0,Y 425.264,Z 157.011,A -85,B 0,C 180,E1 -9688.074,E2 -9688.074} C_VEL
LIN {X 0,Y 425.31,Z 157.002,A -85,B 0,C 180,E1 -9691.367,E2 -9691.367} C_VEL
LIN {X 0,Y 425.271,Z 157.012,A -85,B 0,C 180,E1 -9694.554,E2 -9694.554} C_VEL
LIN {X 0,Y 425.304,Z 157.007,A -85,B 0,C 180,E1 -9696.635,E2 -9696.635} C_VEL
LIN {X 0,Y 425.328,Z 157.006,A -85,B 0,C 180,E1 -9700.365,E2 -9700.365} C_VEL
LIN {X 0,Y 425.388,Z 156.995,A -85,B 0,C 180,E1 -9703.689,E2 -9703.689} C_VEL
LIN {X 0,Y 425.412,Z 156.992,A -85,B 0,C 180,E1 -9707.599,E2 -9707.599} C_VEL
LIN {X 0,Y 425.407,Z 156.992,A -85,B 0,C 180,E1 -9711.45,E2 -9711.45} C_VEL
LIN {X 0,Y 425.526,Z 156.978,A -85,B 0,C 180,E1 -9714.313,E2 -9714.313} C_VEL
LIN {X 0,Y 425.564,Z 156.975,A -85,B 0,C 180,E1 -9718.108,E2 -9718.108} C_VEL
LIN {X 0,Y 425.572,Z 156.974,A -85,B 0,C 180,E1 -9720,E2 -9720} C_VEL
LIN {X 0,Y 425.524,Z 156.976,A -85,B 0,C 180,E1 -9722.84,E2 -9722.84} C_VEL
LIN {X 0,Y 425.47,Z 156.982,A -85,B 0,C 180,E1 -9726.64,E2 -9726.64} C_VEL
LIN {X 0,Y 425.386,Z 157,A -85,B 0,C 180,E1 -9729.51,E2 -9729.51} C_VEL
LIN {X 0,Y 425.395,Z 156.993,A -85,B 0,C 180,E1 -9732.904,E2 -9732.904} C_VEL
LIN {X 0,Y 425.348,Z 156.998,A -85,B 0,C 180,E1 -9736.598,E2 -9736.598} C_VEL
LIN {X 0,Y 425.329,Z 157.004,A -85,B 0,C 180,E1 -9739.635,E2 -9739.635} C_VEL
LIN {X 0,Y 425.289,Z 157.005,A -85,B 0,C 180,E1 -9742.339,E2 -9742.339} C_VEL
LIN {X 0,Y 425.253,Z 157.014,A -85,B 0,C 180,E1 -9745.449,E2 -9745.449} C_VEL
LIN {X 0,Y 425.297,Z 157.008,A -85,B 0,C 180,E1 -9748.857,E2 -9748.857} C_VEL
LIN {X 0,Y 425.247,Z 157.01,A -85,B 0,C 180,E1 -9751.929,E2 -9751.929} C_VEL
LIN {X 0,Y 425.293,Z 157.008,A -85,B 0,C 180,E1 -9755.337,E2 -9755.337} C_VEL
LIN {X 0,Y 425.268,Z 157.015,A -85,B 0,C 180,E1 -9758.902,E2 -9758.902} C_VEL
LIN {X 0,Y 425.264,Z 157.008,A -85,B 0,C 180,E1 -9761.954,E2 -9761.954} C_VEL
LIN {X 0,Y 425.287,Z 157.007,A -85,B 0,C 180,E1 -9765.283,E2 -9765.283} C_VEL
LIN {X 0,Y 425.247,Z 157.016,A -85,B 0,C 180,E1 -9768.618,E2 -9768.618} C_VEL
LIN {X 0,Y 425.267,Z 157.011,A -85,B 0,C 180,E1 -9772.304,E2 -9772.304} C_VEL
LIN {X 0,Y 425.259,Z 157.009,A -85,B 0,C 180,E1 -9775.812,E2 -9775.812} C_VEL
LIN {X 0,Y 425.287,Z 157.01,A -85,B 0,C 180,E1 -9779.24,E2 -9779.24} C_VEL
LIN {X 0,Y 425.241,Z 157.018,A -85,B 0,C 180,E1 -9782.434,E2 -9782.434} C_VEL
LIN {X 0,Y 425.325,Z 157.125,A -85,B 0,C 180,E1 -9783.701,E2 -9783.701} C_VEL
LIN {X 0,Y 427.756,Z 169.538,A -85,B 0,C 180,E1 -9786.52,E2 -9786.52} C_VEL
LIN {X 0,Y 427.786,Z 174.494,A -85,B 0,C 180,E1 -9787.56,E2 -9787.56} C_VEL
LIN {X 0,Y 426.636,Z 193.004,A -85,B 0,C 180,E1 -9791.312,E2 -9791.312} C_VEL
LIN {X 0,Y 426.82,Z 194.703,A -85,B 0,C 180,E1 -9791.414,E2 -9791.414} C_VEL
LIN {X 0,Y 430.353,Z 216.426,A -85,B 0,C 180,E1 -9791.953,E2 -9791.953} C_VEL
LIN {X 0,Y 429.369,Z 301.534,A -85,B 0,C 180,E1 -9793.446,E2 -9793.446} C_VEL
LIN {X 0,Y 428.874,Z 315.302,A -85,B 0,C 180,E1 -9793.885,E2 -9793.885} C_VEL
LIN {X 0,Y 428.305,Z 327.717,A -85,B 0,C 180,E1 -9794.474,E2 -9794.474} C_VEL
LIN {X 0,Y 427.645,Z 339.614,A -85,B 0,C 180,E1 -9795.242,E2 -9795.242} C_VEL
LIN {X 0,Y 426.943,Z 351.379,A -85,B 0,C 180,E1 -9796.22,E2 -9796.22} C_VEL
LIN {X 0,Y 426.4,Z 361.38,A -85,B 0,C 180,E1 -9797.264,E2 -9797.264} C_VEL
LIN {X 0,Y 425.654,Z 371.45,A -85,B 0,C 180,E1 -9798.571,E2 -9798.571} C_VEL
LIN {X 0,Y 425.078,Z 380.311,A -85,B 0,C 180,E1 -9800.002,E2 -9800.002} C_VEL
LIN {X 0,Y 424.649,Z 387.39,A -85,B 0,C 180,E1 -9801.433,E2 -9801.433} C_VEL
LIN {X 0,Y 424.364,Z 393.042,A -85,B 0,C 180,E1 -9802.864,E2 -9802.864} C_VEL
LIN {X 0,Y 424.212,Z 397.482,A -85,B 0,C 180,E1 -9804.294,E2 -9804.294} C_VEL
LIN {X 0,Y 424.206,Z 399.825,A -85,B 0,C 180,E1 -9805.247,E2 -9805.247} C_VEL
LIN {X 0,Y 424.082,Z 401.734,A -85,B 0,C 180,E1 -9806.198,E2 -9806.198} C_VEL
LIN {X 0,Y 424.087,Z 403.19,A -85,B 0,C 180,E1 -9807.149,E2 -9807.149} C_VEL
LIN {X 0,Y 424.122,Z 404.217,A -85,B 0,C 180,E1 -9808.1,E2 -9808.1} C_VEL
LIN {X 0,Y 424.063,Z 405.095,A -85,B 0,C 180,E1 -9809.999,E2 -9809.999} C_VEL
LIN {X 0,Y 424.069,Z 404.914,A -85,B 0,C 180,E1 -9810.949,E2 -9810.949} C_VEL
LIN {X 0,Y 424.122,Z 404.32,A -85,B 0,C 180,E1 -9811.898,E2 -9811.898} C_VEL
LIN {X 0,Y 424.086,Z 403.335,A -85,B 0,C 180,E1 -9812.849,E2 -9812.849} C_VEL
LIN {X 0,Y 424.082,Z 401.952,A -85,B 0,C 180,E1 -9813.8,E2 -9813.8} C_VEL
LIN {X 0,Y 424.244,Z 399.03,A -85,B 0,C 180,E1 -9815.227,E2 -9815.227} C_VEL
LIN {X 0,Y 424.31,Z 395.072,A -85,B 0,C 180,E1 -9816.657,E2 -9816.657} C_VEL
LIN {X 0,Y 424.635,Z 388.991,A -85,B 0,C 180,E1 -9818.326,E2 -9818.326} C_VEL
LIN {X 0,Y 425.032,Z 382.33,A -85,B 0,C 180,E1 -9819.757,E2 -9819.757} C_VEL
LIN {X 0,Y 425.567,Z 374.064,A -85,B 0,C 180,E1 -9821.188,E2 -9821.188} C_VEL
LIN {X 0,Y 426.26,Z 365.609,A -85,B 0,C 180,E1 -9822.376,E2 -9822.376} C_VEL
LIN {X 0,Y 426.901,Z 356.112,A -85,B 0,C 180,E1 -9823.47,E2 -9823.47} C_VEL
LIN {X 0,Y 427.573,Z 344.857,A -85,B 0,C 180,E1 -9824.516,E2 -9824.516} C_VEL
LIN {X 0,Y 428.233,Z 333.58,A -85,B 0,C 180,E1 -9825.344,E2 -9825.344} C_VEL
LIN {X 0,Y 428.991,Z 320.852,A -85,B 0,C 180,E1 -9826.048,E2 -9826.048} C_VEL
LIN {X 0,Y 429.525,Z 307.273,A -85,B 0,C 180,E1 -9826.577,E2 -9826.577} C_VEL
LIN {X 0,Y 429.868,Z 293.551,A -85,B 0,C 180,E1 -9826.899,E2 -9826.899} C_VEL
LIN {X 0,Y 430.797,Z 216.334,A -85,B 0,C 180,E1 -9828.245,E2 -9828.245} C_VEL
LIN {X 0,Y 426.837,Z 192.985,A -85,B 0,C 180,E1 -9828.891,E2 -9828.891} C_VEL
LIN {X 0,Y 427.364,Z 182.607,A -85,B 0,C 180,E1 -9830.931,E2 -9830.931} C_VEL
LIN {X 0,Y 427.99,Z 171.449,A -85,B 0,C 180,E1 -9833.209,E2 -9833.209} C_VEL
LIN {X 0,Y 426.619,Z 163.182,A -85,B 0,C 180,E1 -9835.034,E2 -9835.034} C_VEL
LIN {X 0,Y 425.312,Z 157.066,A -85,B 0,C 180,E1 -9836.496,E2 -9836.496} C_VEL
LIN {X 0,Y 425.267,Z 157.013,A -85,B 0,C 180,E1 -9839.72,E2 -9839.72} C_VEL
LIN {X 0,Y 425.263,Z 157.011,A -85,B 0,C 180,E1 -9843.048,E2 -9843.048} C_VEL
LIN {X 0,Y 425.271,Z 157.012,A -85,B 0,C 180,E1 -9845.926,E2 -9845.926} C_VEL
LIN {X 0,Y 425.251,Z 157.014,A -85,B 0,C 180,E1 -9849.035,E2 -9849.035} C_VEL
LIN {X 0,Y 425.248,Z 157.013,A -85,B 0,C 180,E1 -9852.654,E2 -9852.654} C_VEL
LIN {X 0,Y 425.276,Z 157.014,A -85,B 0,C 180,E1 -9855.282,E2 -9855.282} C_VEL
LIN {X 0,Y 425.239,Z 157.015,A -85,B 0,C 180,E1 -9858.617,E2 -9858.617} C_VEL
LIN {X 0,Y 425.269,Z 157.015,A -85,B 0,C 180,E1 -9861.098,E2 -9861.098} C_VEL
LIN {X 0,Y 425.284,Z 157.009,A -85,B 0,C 180,E1 -9864.662,E2 -9864.662} C_VEL
LIN {X 0,Y 425.242,Z 157.011,A -85,B 0,C 180,E1 -9868.071,E2 -9868.071} C_VEL
LIN {X 0,Y 425.284,Z 157.009,A -85,B 0,C 180,E1 -9871.364,E2 -9871.364} C_VEL
LIN {X 0,Y 425.247,Z 157.013,A -85,B 0,C 180,E1 -9874.551,E2 -9874.551} C_VEL
LIN {X 0,Y 425.28,Z 157.006,A -85,B 0,C 180,E1 -9877.729,E2 -9877.729} C_VEL
LIN {X 0,Y 425.349,Z 156.997,A -85,B 0,C 180,E1 -9880.703,E2 -9880.703} C_VEL
LIN {X 0,Y 425.375,Z 156.993,A -85,B 0,C 180,E1 -9883.687,E2 -9883.687} C_VEL
LIN {X 0,Y 425.399,Z 156.991,A -85,B 0,C 180,E1 -9887.597,E2 -9887.597} C_VEL
LIN {X 0,Y 425.394,Z 156.993,A -85,B 0,C 180,E1 -9891.449,E2 -9891.449} C_VEL
LIN {X 0,Y 425.526,Z 156.978,A -85,B 0,C 180,E1 -9894.312,E2 -9894.312} C_VEL
LIN {X 0,Y 425.554,Z 156.974,A -85,B 0,C 180,E1 -9898.107,E2 -9898.107} C_VEL
LIN {X 0,Y 425.503,Z 156.983,A -85,B 0,C 180,E1 -9900.946,E2 -9900.946} C_VEL
LIN {X 0,Y 425.503,Z 156.979,A -85,B 0,C 180,E1 -9902.84,E2 -9902.84} C_VEL
LIN {X 0,Y 425.525,Z 156.977,A -85,B 0,C 180,E1 -9905.687,E2 -9905.687} C_VEL
LIN {X 0,Y 425.39,Z 156.996,A -85,B 0,C 180,E1 -9908.551,E2 -9908.551} C_VEL
LIN {X 0,Y 425.394,Z 156.998,A -85,B 0,C 180,E1 -9912.402,E2 -9912.402} C_VEL
LIN {X 0,Y 425.373,Z 157,A -85,B 0,C 180,E1 -9916.312,E2 -9916.312} C_VEL
LIN {X 0,Y 425.314,Z 157.006,A -85,B 0,C 180,E1 -9919.635,E2 -9919.635} C_VEL
LIN {X 0,Y 425.274,Z 157.013,A -85,B 0,C 180,E1 -9922.339,E2 -9922.339} C_VEL
LIN {X 0,Y 425.245,Z 157.012,A -85,B 0,C 180,E1 -9925.448,E2 -9925.448} C_VEL
LIN {X 0,Y 425.284,Z 157.012,A -85,B 0,C 180,E1 -9928.858,E2 -9928.858} C_VEL
LIN {X 0,Y 425.315,Z 157.16,A -85,B 0,C 180,E1 -9929.922,E2 -9929.922} C_VEL
LIN {X 0,Y 427.351,Z 167.337,A -85,B 0,C 180,E1 -9932.308,E2 -9932.308} C_VEL
LIN {X 0,Y 427.461,Z 171.385,A -85,B 0,C 180,E1 -9933.189,E2 -9933.189} C_VEL
LIN {X 0,Y 427.045,Z 180.848,A -85,B 0,C 180,E1 -9935.148,E2 -9935.148} C_VEL
LIN {X 0,Y 428.319,Z 187.385,A -85,B 0,C 180,E1 -9935.373,E2 -9935.373} C_VEL
LIN {X 0,Y 430.959,Z 201.891,A -85,B 0,C 180,E1 -9935.769,E2 -9935.769} C_VEL
LIN {X 0,Y 429.755,Z 288.873,A -85,B 0,C 180,E1 -9937.308,E2 -9937.308} C_VEL
LIN {X 0,Y 429.381,Z 302.088,A -85,B 0,C 180,E1 -9937.735,E2 -9937.735} C_VEL
LIN {X 0,Y 428.85,Z 314.717,A -85,B 0,C 180,E1 -9938.334,E2 -9938.334} C_VEL
LIN {X 0,Y 428.187,Z 327.204,A -85,B 0,C 180,E1 -9939.149,E2 -9939.149} C_VEL
LIN {X 0,Y 427.412,Z 338.863,A -85,B 0,C 180,E1 -9940.131,E2 -9940.131} C_VEL
LIN {X 0,Y 426.714,Z 349.019,A -85,B 0,C 180,E1 -9941.208,E2 -9941.208} C_VEL
LIN {X 0,Y 426.089,Z 357.922,A -85,B 0,C 180,E1 -9942.371,E2 -9942.371} C_VEL
LIN {X 0,Y 425.468,Z 366.296,A -85,B 0,C 180,E1 -9943.71,E2 -9943.71} C_VEL
LIN {X 0,Y 424.964,Z 373.113,A -85,B 0,C 180,E1 -9945.049,E2 -9945.049} C_VEL
LIN {X 0,Y 424.634,Z 378.665,A -85,B 0,C 180,E1 -9946.395,E2 -9946.395} C_VEL
LIN {X 0,Y 424.429,Z 383.141,A -85,B 0,C 180,E1 -9947.753,E2 -9947.753} C_VEL
LIN {X 0,Y 424.24,Z 386.644,A -85,B 0,C 180,E1 -9949.12,E2 -9949.12} C_VEL
LIN {X 0,Y 424.003,Z 389.933,A -85,B 0,C 180,E1 -9950.962,E2 -9950.962} C_VEL
LIN {X 0,Y 423.902,Z 391.571,A -85,B 0,C 180,E1 -9952.731,E2 -9952.731} C_VEL
LIN {X 0,Y 423.895,Z 391.836,A -85,B 0,C 180,E1 -9954.531,E2 -9954.531} C_VEL
LIN {X 0,Y 423.914,Z 390.988,A -85,B 0,C 180,E1 -9955.989,E2 -9955.989} C_VEL
LIN {X 0,Y 424.034,Z 388.795,A -85,B 0,C 180,E1 -9957.701,E2 -9957.701} C_VEL
LIN {X 0,Y 424.242,Z 385.947,A -85,B 0,C 180,E1 -9959.101,E2 -9959.101} C_VEL
LIN {X 0,Y 424.461,Z 381.283,A -85,B 0,C 180,E1 -9960.763,E2 -9960.763} C_VEL
LIN {X 0,Y 424.787,Z 375.102,A -85,B 0,C 180,E1 -9962.404,E2 -9962.404} C_VEL
LIN {X 0,Y 425.174,Z 368.661,A -85,B 0,C 180,E1 -9963.759,E2 -9963.759} C_VEL
LIN {X 0,Y 425.604,Z 361.833,A -85,B 0,C 180,E1 -9964.94,E2 -9964.94} C_VEL
LIN {X 0,Y 426.231,Z 352.201,A -85,B 0,C 180,E1 -9966.304,E2 -9966.304} C_VEL
LIN {X 0,Y 426.903,Z 342.371,A -85,B 0,C 180,E1 -9967.417,E2 -9967.417} C_VEL
LIN {X 0,Y 427.586,Z 331.365,A -85,B 0,C 180,E1 -9968.424,E2 -9968.424} C_VEL
LIN {X 0,Y 428.234,Z 319.114,A -85,B 0,C 180,E1 -9969.301,E2 -9969.301} C_VEL
LIN {X 0,Y 428.826,Z 306.023,A -85,B 0,C 180,E1 -9969.995,E2 -9969.995} C_VEL
LIN {X 0,Y 429.231,Z 292.898,A -85,B 0,C 180,E1 -9970.482,E2 -9970.482} C_VEL
LIN {X 0,Y 429.512,Z 277.77,A -85,B 0,C 180,E1 -9970.806,E2 -9970.806} C_VEL
LIN {X 0,Y 429.696,Z 263.255,A -85,B 0,C 180,E1 -9971.055,E2 -9971.055} C_VEL
LIN {X 0,Y 429.148,Z 257.447,A -85,B 0,C 180,E1 -9971.178,E2 -9971.178} C_VEL
LIN {X 0,Y 423.783,Z 238.767,A -85,B 0,C 180,E1 -9971.72,E2 -9971.72} C_VEL
LIN {X 0,Y 423.205,Z 232.959,A -85,B 0,C 180,E1 -9971.848,E2 -9971.848} C_VEL
LIN {X 0,Y 423.563,Z 201.639,A -85,B 0,C 180,E1 -9972.401,E2 -9972.401} C_VEL
LIN {X 0,Y 419.86,Z 181.358,A -85,B 0,C 180,E1 -9972.953,E2 -9972.953} C_VEL
LIN {X 0,Y 419.829,Z 180.171,A -85,B 0,C 180,E1 -9973.124,E2 -9973.124} C_VEL
LIN {X 0,Y 420.485,Z 169.642,A -85,B 0,C 180,E1 -9975.482,E2 -9975.482} C_VEL
LIN {X 0,Y 418.398,Z 158.216,A -85,B 0,C 180,E1 -9978.25,E2 -9978.25} C_VEL
LIN {X 0,Y 418.323,Z 157.879,A -85,B 0,C 180,E1 -9978.616,E2 -9978.616} C_VEL
LIN {X 0,Y 418.49,Z 157.855,A -85,B 0,C 180,E1 -9982.28,E2 -9982.28} C_VEL
LIN {X 0,Y 418.51,Z 157.853,A -85,B 0,C 180,E1 -9984.218,E2 -9984.218} C_VEL
LIN {X 0,Y 418.539,Z 157.85,A -85,B 0,C 180,E1 -9988.076,E2 -9988.076} C_VEL
LIN {X 0,Y 418.668,Z 157.834,A -85,B 0,C 180,E1 -9990.001,E2 -9990.001} C_VEL
LIN {X 0,Y 418.499,Z 157.851,A -85,B 0,C 180,E1 -9992.889,E2 -9992.889} C_VEL
LIN {X 0,Y 418.503,Z 157.856,A -85,B 0,C 180,E1 -9995.784,E2 -9995.784} C_VEL
LIN {X 0,Y 418.376,Z 157.866,A -85,B 0,C 180,E1 -9998.696,E2 -9998.696} C_VEL
LIN {X 0,Y 418.314,Z 157.879,A -85,B 0,C 180,E1 -10001.632,E2 -10001.632} C_VEL
LIN {X 0,Y 418.301,Z 157.876,A -85,B 0,C 180,E1 -10004.598,E2 -10004.598} C_VEL
LIN {X 0,Y 418.279,Z 157.883,A -85,B 0,C 180,E1 -10007.605,E2 -10007.605} C_VEL
LIN {X 0,Y 418.249,Z 157.883,A -85,B 0,C 180,E1 -10010.664,E2 -10010.664} C_VEL
LIN {X 0,Y 418.284,Z 157.879,A -85,B 0,C 180,E1 -10013.782,E2 -10013.782} C_VEL
LIN {X 0,Y 418.31,Z 157.881,A -85,B 0,C 180,E1 -10017.071,E2 -10017.071} C_VEL
LIN {X 0,Y 418.244,Z 157.883,A -85,B 0,C 180,E1 -10020.273,E2 -10020.273} C_VEL
LIN {X 0,Y 418.246,Z 157.883,A -85,B 0,C 180,E1 -10023.678,E2 -10023.678} C_VEL
LIN {X 0,Y 418.239,Z 157.887,A -85,B 0,C 180,E1 -10027.225,E2 -10027.225} C_VEL
LIN {X 0,Y 418.244,Z 157.883,A -85,B 0,C 180,E1 -10029.683,E2 -10029.683} C_VEL
LIN {X 0,Y 418.229,Z 157.886,A -85,B 0,C 180,E1 -10032.322,E2 -10032.322} C_VEL
LIN {X 0,Y 418.235,Z 157.887,A -85,B 0,C 180,E1 -10035.109,E2 -10035.109} C_VEL
LIN {X 0,Y 418.233,Z 157.884,A -85,B 0,C 180,E1 -10037.767,E2 -10037.767} C_VEL
LIN {X 0,Y 418.237,Z 157.883,A -85,B 0,C 180,E1 -10041.557,E2 -10041.557} C_VEL
LIN {X 0,Y 418.258,Z 157.882,A -85,B 0,C 180,E1 -10045.159,E2 -10045.159} C_VEL
LIN {X 0,Y 418.245,Z 157.882,A -85,B 0,C 180,E1 -10047.472,E2 -10047.472} C_VEL
LIN {X 0,Y 418.263,Z 157.882,A -85,B 0,C 180,E1 -10050.897,E2 -10050.897} C_VEL
LIN {X 0,Y 418.236,Z 157.888,A -85,B 0,C 180,E1 -10054.094,E2 -10054.094} C_VEL
LIN {X 0,Y 418.237,Z 157.883,A -85,B 0,C 180,E1 -10057.264,E2 -10057.264} C_VEL
LIN {X 0,Y 418.283,Z 157.883,A -85,B 0,C 180,E1 -10060.365,E2 -10060.365} C_VEL
LIN {X 0,Y 418.316,Z 157.874,A -85,B 0,C 180,E1 -10063.405,E2 -10063.405} C_VEL
LIN {X 0,Y 418.347,Z 157.87,A -85,B 0,C 180,E1 -10067,E2 -10067} C_VEL
LIN {X 0,Y 418.335,Z 157.875,A -85,B 0,C 180,E1 -10070.329,E2 -10070.329} C_VEL
LIN {X 0,Y 418.441,Z 157.859,A -85,B 0,C 180,E1 -10073.249,E2 -10073.249} C_VEL
LIN {X 0,Y 418.318,Z 157.874,A -85,B 0,C 180,E1 -10075.182,E2 -10075.182} C_VEL
LIN {X 0,Y 418.533,Z 157.851,A -85,B 0,C 180,E1 -10078.076,E2 -10078.076} C_VEL
LIN {X 0,Y 418.407,Z 157.863,A -85,B 0,C 180,E1 -10080.963,E2 -10080.963} C_VEL
LIN {X 0,Y 418.481,Z 157.853,A -85,B 0,C 180,E1 -10082.888,E2 -10082.888} C_VEL
LIN {X 0,Y 418.436,Z 157.859,A -85,B 0,C 180,E1 -10086.752,E2 -10086.752} C_VEL
LIN {X 0,Y 418.327,Z 157.878,A -85,B 0,C 180,E1 -10089.672,E2 -10089.672} C_VEL
LIN {X 0,Y 418.348,Z 157.872,A -85,B 0,C 180,E1 -10093.001,E2 -10093.001} C_VEL
LIN {X 0,Y 418.307,Z 157.876,A -85,B 0,C 180,E1 -10096.732,E2 -10096.732} C_VEL
LIN {X 0,Y 418.271,Z 157.882,A -85,B 0,C 180,E1 -10099.789,E2 -10099.789} C_VEL
LIN {X 0,Y 418.229,Z 157.886,A -85,B 0,C 180,E1 -10102.737,E2 -10102.737} C_VEL
LIN {X 0,Y 418.212,Z 157.887,A -85,B 0,C 180,E1 -10105.908,E2 -10105.908} C_VEL
